Yaskawa INFORM job: aprem2TRJ2.JBI

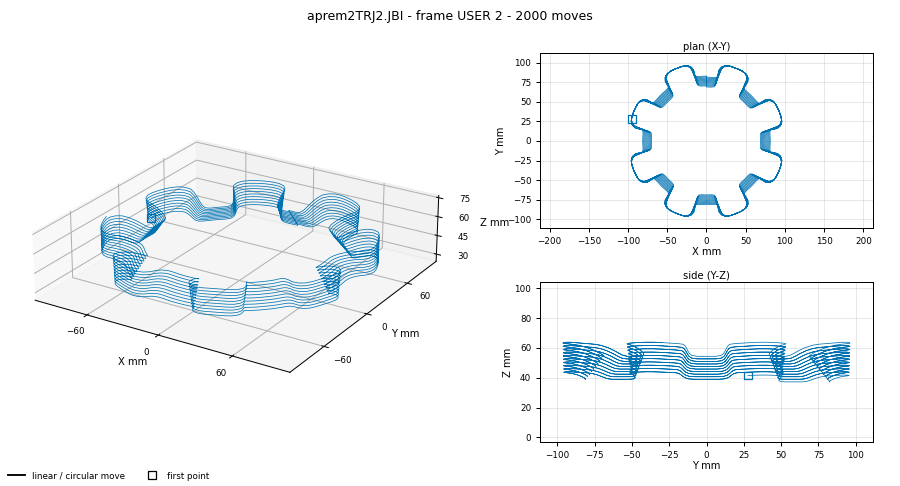
[picture p0: tool path of aprem2TRJ2.JBI in frame USER 2, 2000 of 2000 moves have a stored position in this frame; points joined in program order, loops and branches not executed]
/JOB
//NAME aprem2TRJ2
//POS
///NPOS 2000,0,2000,0,0,0
///USER 2
///TOOL 1
///POSTYPE USER
///RECTAN
///RCONF 1,0,0,0,0,0,0,0,0,0,0,0,0,0,0,0,0,0,0,0,0,0,0,0
C00000=-95.500,27.752,41.515,179.9573,-1.4576,0.0000
C00001=-94.679,31.992,41.678,179.9802,-0.0621,0.0000
C00002=-93.214,36.189,41.785,179.9968,-0.0083,0.0000
C00003=-91.502,40.323,41.785,179.9964,-0.0081,0.0000
C00004=-89.570,44.326,41.678,179.9701,-0.0579,0.0000
C00005=-87.153,47.905,41.515,178.9994,-1.0610,0.0000
C00006=-83.964,50.341,41.355,177.9940,-1.0426,0.0000
C00007=-80.606,51.270,41.159,176.0647,-0.0633,0.0000
C00008=-77.545,50.645,40.789,176.2827,1.1365,0.0000
C00009=-74.511,49.565,40.048,179.1830,0.2954,0.0000
C00010=-71.724,48.673,39.090,-174.7304,-1.4587,0.0000
C00011=-69.261,48.447,38.165,-161.9042,-0.3246,0.0000
C00012=-66.868,49.465,37.495,-150.0988,20.4873,0.0000
C00013=-64.059,52.288,37.229,-152.5931,29.6910,0.0000
C00014=-61.349,55.398,37.217,-152.6199,30.0136,0.0000
C00015=-58.451,58.451,37.225,-151.2604,28.7392,0.0000
C00016=-55.398,61.349,37.217,-149.9866,27.3805,0.0000
C00017=-52.288,64.059,37.229,-150.3100,27.4077,0.0000
C00018=-49.465,66.868,37.495,-159.5118,29.9009,0.0000
C00019=-48.447,69.261,38.165,179.6754,18.0958,0.0000
C00020=-48.673,71.724,39.090,178.5413,5.2696,0.0000
C00021=-49.565,74.511,40.048,-179.7046,-0.8170,0.0000
C00022=-50.645,77.545,40.789,-178.8635,-3.7173,0.0000
C00023=-51.270,80.606,41.159,179.9367,-3.9353,0.0000
C00024=-50.341,83.964,41.355,178.9574,-2.0060,0.0000
C00025=-47.905,87.153,41.515,178.9390,-1.0006,0.0000
C00026=-44.326,89.570,41.678,179.9421,-0.0299,0.0000
C00027=-40.323,91.502,41.785,179.9919,-0.0036,0.0000
C00028=-36.189,93.214,41.785,179.9917,-0.0032,0.0000
C00029=-31.992,94.679,41.678,179.9379,-0.0198,0.0000
C00030=-27.752,95.500,41.515,178.5424,-0.0427,0.0000
C00031=-23.775,94.968,41.355,177.8447,0.6817,0.0000
C00032=-20.743,93.250,41.159,177.1705,2.7402,0.0000
C00033=-19.021,90.644,40.789,178.1721,3.4318,0.0000
C00034=-17.640,87.735,40.048,179.6311,0.7865,0.0000
C00035=-16.299,85.134,39.090,-177.2970,-4.7574,0.0000
C00036=-14.718,83.232,38.165,-167.2077,-13.2282,0.0000
C00037=-12.305,82.260,37.495,-146.1451,-8.1050,0.0000
C00038=-8.324,82.270,37.229,-142.4105,2.0911,0.0000
C00039=-4.208,82.553,37.217,-142.2353,2.4190,0.0000
C00040=0.000,82.662,37.225,-142.2055,0.0004,0.0000
C00041=0.000,81.307,38.958,-141.7581,0.0003,0.0000
C00042=4.084,81.202,38.949,-141.7876,-2.4412,0.0000
C00043=8.115,80.931,38.962,-141.9747,-1.8578,0.0000
C00044=12.050,80.963,39.253,-146.2950,9.3084,0.0000
C00045=14.402,82.041,39.987,-169.0753,12.6711,0.0000
C00046=15.932,84.113,41.004,-178.0957,3.7141,0.0000
C00047=17.234,86.943,42.060,179.2930,-1.6621,0.0000
C00048=18.580,90.119,42.880,177.9599,-4.2630,0.0000
C00049=20.259,92.987,43.289,176.7690,-3.4884,0.0000
C00050=23.317,94.913,43.506,177.4450,-0.9091,0.0000
C00051=27.389,95.566,43.684,178.3657,0.0207,0.0000
C00052=31.762,94.755,43.864,179.9236,0.0242,0.0000
C00053=36.110,93.244,43.984,179.9901,0.0038,0.0000
C00054=40.400,91.468,43.984,179.9903,0.0044,0.0000
C00055=44.543,89.461,43.864,179.9289,0.0369,0.0000
C00056=48.209,86.942,43.684,178.8296,1.1411,0.0000
C00057=50.626,83.601,43.506,178.8351,2.4492,0.0000
C00058=51.426,80.077,43.289,-179.8173,4.7459,0.0000
C00059=50.586,76.861,42.880,-178.4237,4.4542,0.0000
C00060=49.291,73.664,42.060,-179.3244,1.6751,0.0000
C00061=48.211,70.742,41.004,178.7173,-3.9706,0.0000
C00062=47.828,68.195,39.987,178.7113,-16.4605,0.0000
C00063=48.729,65.770,39.253,-160.4159,-30.4372,0.0000
C00064=51.488,62.965,38.962,-150.0628,-27.9244,0.0000
C00065=54.531,60.307,38.949,-149.5942,-27.7685,0.0000
C00066=57.493,57.493,38.958,-150.8703,-29.1301,0.0000
C00067=60.306,54.531,38.949,-152.2311,-30.4055,0.0000
C00068=62.965,51.488,38.962,-152.0747,-29.9361,0.0000
C00069=65.770,48.729,39.253,-149.5629,-19.5850,0.0000
C00070=68.195,47.828,39.987,-163.5395,1.2887,0.0000
C00071=70.742,48.211,41.004,-176.0294,1.2827,0.0000
C00072=73.664,49.291,42.060,178.3249,-0.6756,0.0000
C00073=76.861,50.586,42.880,175.5458,-1.5763,0.0000
C00074=80.077,51.426,43.289,175.2541,-0.1827,0.0000
C00075=83.601,50.626,43.506,177.5508,1.1649,0.0000
C00076=86.942,48.209,43.684,178.8589,1.1704,0.0000
C00077=89.461,44.543,43.864,179.9631,0.0711,0.0000
C00078=91.468,40.400,43.984,179.9956,0.0097,0.0000
C00079=93.244,36.110,43.984,179.9962,0.0099,0.0000
C00080=94.755,31.762,43.864,179.9758,0.0764,0.0000
C00081=95.566,27.389,43.684,179.9793,1.6343,0.0000
C00082=94.913,23.317,43.506,-179.0909,2.5550,0.0000
C00083=92.987,20.259,43.289,-176.5116,3.2310,0.0000
C00084=90.119,18.580,42.880,-175.7370,2.0401,0.0000
C00085=86.943,17.234,42.060,-178.3379,0.7070,0.0000
C00086=84.113,15.932,41.004,176.2859,-1.9043,0.0000
C00087=82.041,14.402,39.987,167.3289,-10.9247,0.0000
C00088=80.963,12.050,39.253,170.6916,-33.7050,0.0000
C00089=80.931,8.115,38.962,-178.1422,-38.0253,0.0000
C00090=81.202,4.084,38.949,-177.5588,-38.2124,0.0000
C00091=81.307,0.000,38.958,179.9997,-38.2419,0.0000
C00092=81.202,-4.084,38.949,177.5593,-38.2124,0.0000
C00093=80.931,-8.116,38.962,178.1440,-38.0251,0.0000
C00094=80.963,-12.050,39.253,-170.6925,-33.7054,0.0000
C00095=82.041,-14.402,39.987,-167.3289,-10.9247,0.0000
C00096=84.113,-15.932,41.004,-176.2859,-1.9043,0.0000
C00097=86.943,-17.234,42.060,178.3379,0.7070,0.0000
C00098=90.119,-18.580,42.880,175.7370,2.0401,0.0000
C00099=92.987,-20.259,43.289,176.5116,3.2310,0.0000
C00100=94.913,-23.317,43.506,179.0909,2.5550,0.0000
C00101=95.566,-27.389,43.684,-179.9793,1.6343,0.0000
C00102=94.755,-31.762,43.864,-179.9758,0.0764,0.0000
C00103=93.244,-36.110,43.984,-179.9962,0.0099,0.0000
C00104=91.468,-40.400,43.984,-179.9956,0.0097,0.0000
C00105=89.461,-44.543,43.864,-179.9631,0.0711,0.0000
C00106=86.942,-48.209,43.684,-178.8589,1.1704,0.0000
C00107=83.601,-50.626,43.506,-177.5508,1.1649,0.0000
C00108=80.077,-51.426,43.289,-175.2541,-0.1827,0.0000
C00109=76.861,-50.586,42.880,-175.5458,-1.5763,0.0000
C00110=73.664,-49.291,42.060,-178.3249,-0.6756,0.0000
C00111=70.742,-48.211,41.004,176.0294,1.2827,0.0000
C00112=68.195,-47.828,39.987,163.5395,1.2887,0.0000
C00113=65.770,-48.729,39.253,149.5628,-19.5841,0.0000
C00114=62.965,-51.488,38.962,152.0756,-29.9372,0.0000
C00115=60.307,-54.531,38.949,152.2315,-30.4058,0.0000
C00116=57.493,-57.493,38.958,150.8699,-29.1297,0.0000
C00117=54.531,-60.306,38.949,149.5945,-27.7689,0.0000
C00118=51.488,-62.965,38.962,150.0639,-27.9253,0.0000
C00119=48.729,-65.770,39.253,160.4150,-30.4371,0.0000
C00120=47.828,-68.195,39.987,-178.7113,-16.4605,0.0000
C00121=48.211,-70.742,41.004,-178.7173,-3.9706,0.0000
C00122=49.291,-73.664,42.060,179.3244,1.6751,0.0000
C00123=50.586,-76.861,42.880,178.4237,4.4542,0.0000
C00124=51.426,-80.077,43.289,179.8173,4.7459,0.0000
C00125=50.626,-83.601,43.506,-178.8351,2.4492,0.0000
C00126=48.209,-86.942,43.684,-178.8296,1.1411,0.0000
C00127=44.543,-89.461,43.864,-179.9289,0.0369,0.0000
C00128=40.400,-91.468,43.984,-179.9903,0.0044,0.0000
C00129=36.110,-93.244,43.984,-179.9901,0.0038,0.0000
C00130=31.762,-94.755,43.864,-179.9236,0.0242,0.0000
C00131=27.389,-95.566,43.684,-178.3657,0.0207,0.0000
C00132=23.317,-94.913,43.506,-177.4450,-0.9091,0.0000
C00133=20.259,-92.987,43.289,-176.7690,-3.4884,0.0000
C00134=18.580,-90.119,42.880,-177.9599,-4.2630,0.0000
C00135=17.234,-86.943,42.060,-179.2930,-1.6621,0.0000
C00136=15.932,-84.113,41.004,178.0957,3.7141,0.0000
C00137=14.402,-82.041,39.987,169.0753,12.6711,0.0000
C00138=12.050,-80.963,39.253,146.2950,9.3084,0.0000
C00139=8.115,-80.931,38.962,141.9747,-1.8578,0.0000
C00140=4.084,-81.202,38.949,141.7876,-2.4412,0.0000
C00141=0.000,-81.307,38.958,141.7581,0.0003,0.0000
C00142=0.000,-81.307,38.958,141.7581,0.0003,0.0000
C00143=-4.084,-81.202,38.949,141.7876,2.4407,0.0000
C00144=-8.116,-80.931,38.962,141.9749,1.8560,0.0000
C00145=-12.050,-80.963,39.253,146.2946,-9.3075,0.0000
C00146=-14.402,-82.041,39.987,169.0753,-12.6711,0.0000
C00147=-15.932,-84.113,41.004,178.0957,-3.7141,0.0000
C00148=-17.234,-86.943,42.060,-179.2930,1.6621,0.0000
C00149=-18.580,-90.119,42.880,-177.9599,4.2630,0.0000
C00150=-20.259,-92.987,43.289,-176.7690,3.4884,0.0000
C00151=-23.317,-94.913,43.506,-177.4450,0.9091,0.0000
C00152=-27.389,-95.566,43.684,-178.3657,-0.0207,0.0000
C00153=-31.762,-94.755,43.864,-179.9236,-0.0242,0.0000
C00154=-36.110,-93.244,43.984,-179.9901,-0.0038,0.0000
C00155=-40.400,-91.468,43.984,-179.9903,-0.0044,0.0000
C00156=-44.543,-89.461,43.864,-179.9289,-0.0369,0.0000
C00157=-48.209,-86.942,43.684,-178.8296,-1.1411,0.0000
C00158=-50.626,-83.601,43.506,-178.8351,-2.4492,0.0000
C00159=-51.426,-80.077,43.289,179.8173,-4.7459,0.0000
C00160=-50.586,-76.861,42.880,178.4237,-4.4542,0.0000
C00161=-49.291,-73.664,42.060,179.3244,-1.6751,0.0000
C00162=-48.211,-70.742,41.004,-178.7173,3.9706,0.0000
C00163=-47.828,-68.195,39.987,-178.7113,16.4605,0.0000
C00164=-48.729,-65.770,39.253,160.4159,30.4372,0.0000
C00165=-51.488,-62.965,38.962,150.0628,27.9244,0.0000
C00166=-54.531,-60.307,38.949,149.5942,27.7685,0.0000
C00167=-57.493,-57.493,38.958,150.8703,29.1301,0.0000
C00168=-60.306,-54.531,38.949,152.2311,30.4055,0.0000
C00169=-62.965,-51.488,38.962,152.0747,29.9361,0.0000
C00170=-65.770,-48.729,39.253,149.5629,19.5850,0.0000
C00171=-68.195,-47.828,39.987,163.5395,-1.2887,0.0000
C00172=-70.742,-48.211,41.004,176.0294,-1.2827,0.0000
C00173=-73.664,-49.291,42.060,-178.3249,0.6756,0.0000
C00174=-76.861,-50.586,42.880,-175.5458,1.5763,0.0000
C00175=-80.077,-51.426,43.289,-175.2541,0.1827,0.0000
C00176=-83.601,-50.626,43.506,-177.5508,-1.1649,0.0000
C00177=-86.942,-48.209,43.684,-178.8589,-1.1704,0.0000
C00178=-89.461,-44.543,43.864,-179.9631,-0.0711,0.0000
C00179=-91.468,-40.400,43.984,-179.9956,-0.0097,0.0000
C00180=-93.244,-36.110,43.984,-179.9962,-0.0099,0.0000
C00181=-94.755,-31.762,43.864,-179.9758,-0.0764,0.0000
C00182=-95.566,-27.389,43.684,-179.9793,-1.6343,0.0000
C00183=-94.913,-23.317,43.506,179.0909,-2.5550,0.0000
C00184=-92.987,-20.259,43.289,176.5116,-3.2310,0.0000
C00185=-90.119,-18.580,42.880,175.7370,-2.0401,0.0000
C00186=-86.943,-17.234,42.060,178.3379,-0.7070,0.0000
C00187=-84.113,-15.932,41.004,-176.2859,1.9043,0.0000
C00188=-82.041,-14.402,39.987,-167.3289,10.9247,0.0000
C00189=-80.963,-12.050,39.253,-170.6916,33.7050,0.0000
C00190=-80.931,-8.115,38.962,178.1422,38.0253,0.0000
C00191=-81.202,-4.084,38.949,177.5588,38.2124,0.0000
C00192=-81.307,0.000,38.958,-179.9997,38.2419,0.0000
C00193=-81.202,4.084,38.949,-177.5593,38.2124,0.0000
C00194=-80.931,8.116,38.962,-178.1440,38.0251,0.0000
C00195=-80.963,12.050,39.253,170.6925,33.7054,0.0000
C00196=-82.041,14.402,39.987,167.3289,10.9247,0.0000
C00197=-84.113,15.932,41.004,176.2859,1.9043,0.0000
C00198=-86.943,17.234,42.060,-178.3379,-0.7070,0.0000
C00199=-90.119,18.580,42.880,-175.7370,-2.0401,0.0000
C00200=-92.987,20.259,43.289,-176.5116,-3.2310,0.0000
C00201=-94.913,23.317,43.506,-179.0909,-2.5550,0.0000
C00202=-95.566,27.389,43.684,179.9793,-1.6343,0.0000
C00203=-94.755,31.762,43.864,179.9758,-0.0764,0.0000
C00204=-93.244,36.110,43.984,179.9962,-0.0099,0.0000
C00205=-91.468,40.400,43.984,179.9956,-0.0097,0.0000
C00206=-89.461,44.543,43.864,179.9631,-0.0711,0.0000
C00207=-86.942,48.209,43.684,178.8589,-1.1704,0.0000
C00208=-83.601,50.626,43.506,177.5508,-1.1649,0.0000
C00209=-80.077,51.426,43.289,175.2541,0.1827,0.0000
C00210=-76.861,50.586,42.880,175.5458,1.5763,0.0000
C00211=-73.664,49.291,42.060,178.3249,0.6756,0.0000
C00212=-70.742,48.211,41.004,-176.0294,-1.2827,0.0000
C00213=-68.195,47.828,39.987,-163.5395,-1.2887,0.0000
C00214=-65.770,48.729,39.253,-149.5628,19.5841,0.0000
C00215=-62.965,51.488,38.962,-152.0756,29.9372,0.0000
C00216=-60.307,54.531,38.949,-152.2315,30.4058,0.0000
C00217=-57.493,57.493,38.958,-150.8699,29.1297,0.0000
C00218=-54.531,60.306,38.949,-149.5945,27.7689,0.0000
C00219=-51.488,62.965,38.962,-150.0639,27.9253,0.0000
C00220=-48.729,65.770,39.253,-160.4150,30.4371,0.0000
C00221=-47.828,68.195,39.987,178.7113,16.4605,0.0000
C00222=-48.211,70.742,41.004,178.7173,3.9706,0.0000
C00223=-49.291,73.664,42.060,-179.3244,-1.6751,0.0000
C00224=-50.586,76.861,42.880,-178.4237,-4.4542,0.0000
C00225=-51.426,80.077,43.289,-179.8173,-4.7459,0.0000
C00226=-50.626,83.601,43.506,178.8351,-2.4492,0.0000
C00227=-48.209,86.942,43.684,178.8296,-1.1411,0.0000
C00228=-44.543,89.461,43.864,179.9289,-0.0369,0.0000
C00229=-40.400,91.468,43.984,179.9903,-0.0044,0.0000
C00230=-36.110,93.244,43.984,179.9901,-0.0038,0.0000
C00231=-31.762,94.755,43.864,179.9236,-0.0242,0.0000
C00232=-27.389,95.566,43.684,178.3657,-0.0207,0.0000
C00233=-23.317,94.913,43.506,177.4450,0.9091,0.0000
C00234=-20.259,92.987,43.289,176.7690,3.4884,0.0000
C00235=-18.580,90.119,42.880,177.9599,4.2630,0.0000
C00236=-17.234,86.943,42.060,179.2930,1.6621,0.0000
C00237=-15.932,84.113,41.004,-178.0957,-3.7141,0.0000
C00238=-14.402,82.041,39.987,-169.0753,-12.6711,0.0000
C00239=-12.050,80.963,39.253,-146.2946,-9.3075,0.0000
C00240=-8.116,80.931,38.962,-141.9749,1.8560,0.0000
C00241=-4.084,81.202,38.949,-141.7876,2.4407,0.0000
C00242=0.000,81.307,38.958,-141.7581,0.0003,0.0000
C00243=0.000,79.940,40.681,-141.3945,0.0003,0.0000
C00244=3.959,79.840,40.672,-141.4236,-2.4543,0.0000
C00245=7.905,79.580,40.686,-141.6255,-1.5989,0.0000
C00246=11.791,79.654,41.003,-146.5959,10.4668,0.0000
C00247=14.083,80.839,41.802,-170.8088,11.8957,0.0000
C00248=15.561,83.082,42.912,-178.7432,2.6994,0.0000
C00249=16.825,86.143,44.068,179.0449,-2.4598,0.0000
C00250=18.134,89.588,44.968,177.8329,-5.0059,0.0000
C00251=19.771,92.721,45.418,176.4774,-4.2024,0.0000
C00252=22.856,94.857,45.657,177.0847,-1.1491,0.0000
C00253=27.022,95.633,45.852,178.2015,-0.0057,0.0000
C00254=31.529,94.831,46.051,179.9101,0.0282,0.0000
C00255=36.031,93.275,46.182,179.9885,0.0043,0.0000
C00256=40.478,91.433,46.182,179.9888,0.0050,0.0000
C00257=44.762,89.350,46.051,179.9165,0.0436,0.0000
C00258=48.515,86.730,45.852,178.7321,1.2760,0.0000
C00259=50.913,83.236,45.657,178.7496,2.8735,0.0000
C00260=51.583,79.544,45.418,-179.5172,5.4544,0.0000
C00261=50.526,76.172,44.968,-177.9852,5.0686,0.0000
C00262=49.015,72.810,44.068,-178.9351,2.4144,0.0000
C00263=47.744,69.752,42.912,178.9787,-2.7968,0.0000
C00264=47.203,67.120,41.802,178.0217,-14.7549,0.0000
C00265=47.986,64.662,41.003,-161.4435,-30.8352,0.0000
C00266=50.682,61.862,40.686,-149.9004,-28.3778,0.0000
C00267=53.655,59.255,40.672,-149.2767,-28.0885,0.0000
C00268=56.526,56.526,40.681,-150.5516,-29.4487,0.0000
C00269=59.255,53.656,40.672,-151.9113,-30.7231,0.0000
C00270=61.862,50.682,40.686,-151.6213,-30.0984,0.0000
C00271=64.662,47.986,41.003,-149.1649,-18.5575,0.0000
C00272=67.120,47.203,41.802,-165.2451,1.9783,0.0000
C00273=69.752,47.744,42.912,-177.2032,1.0213,0.0000
C00274=72.810,49.015,44.068,177.5856,-1.0649,0.0000
C00275=76.172,50.526,44.968,174.9314,-2.0148,0.0000
C00276=79.544,51.583,45.418,174.5456,-0.4828,0.0000
C00277=83.236,50.913,45.657,177.1265,1.2504,0.0000
C00278=86.730,48.515,45.852,178.7240,1.2679,0.0000
C00279=89.350,44.762,46.051,179.9564,0.0835,0.0000
C00280=91.433,40.478,46.182,179.9950,0.0112,0.0000
C00281=93.275,36.031,46.182,179.9957,0.0115,0.0000
C00282=94.831,31.529,46.051,179.9718,0.0899,0.0000
C00283=95.633,27.022,45.852,-179.9943,1.7985,0.0000
C00284=94.857,22.856,45.657,-178.8509,2.9153,0.0000
C00285=92.721,19.771,45.418,-175.7976,3.5226,0.0000
C00286=89.588,18.134,44.968,-174.9941,2.1671,0.0000
C00287=86.143,16.825,44.068,-177.5402,0.9551,0.0000
C00288=83.082,15.561,42.912,177.3006,-1.2568,0.0000
C00289=80.839,14.083,41.802,168.1043,-9.1912,0.0000
C00290=79.654,11.791,41.003,169.5332,-33.4041,0.0000
C00291=79.580,7.905,40.686,-178.4011,-38.3745,0.0000
C00292=79.840,3.959,40.672,-177.5457,-38.5764,0.0000
C00293=79.940,0.000,40.681,179.9997,-38.6055,0.0000
C00294=79.840,-3.959,40.672,177.5462,-38.5764,0.0000
C00295=79.580,-7.905,40.686,178.4031,-38.3743,0.0000
C00296=79.654,-11.792,41.003,-169.5340,-33.4045,0.0000
C00297=80.839,-14.083,41.802,-168.1043,-9.1912,0.0000
C00298=83.082,-15.561,42.912,-177.3006,-1.2568,0.0000
C00299=86.143,-16.825,44.068,177.5402,0.9551,0.0000
C00300=89.588,-18.134,44.968,174.9941,2.1671,0.0000
C00301=92.721,-19.771,45.418,175.7976,3.5226,0.0000
C00302=94.857,-22.856,45.657,178.8509,2.9153,0.0000
C00303=95.633,-27.022,45.852,179.9943,1.7985,0.0000
C00304=94.831,-31.529,46.051,-179.9718,0.0899,0.0000
C00305=93.275,-36.031,46.182,-179.9957,0.0115,0.0000
C00306=91.433,-40.478,46.182,-179.9950,0.0112,0.0000
C00307=89.350,-44.762,46.051,-179.9564,0.0835,0.0000
C00308=86.730,-48.515,45.852,-178.7240,1.2679,0.0000
C00309=83.236,-50.913,45.657,-177.1265,1.2504,0.0000
C00310=79.544,-51.583,45.418,-174.5456,-0.4828,0.0000
C00311=76.172,-50.526,44.968,-174.9314,-2.0148,0.0000
C00312=72.810,-49.015,44.068,-177.5856,-1.0649,0.0000
C00313=69.752,-47.744,42.912,177.2032,1.0213,0.0000
C00314=67.120,-47.203,41.802,165.2451,1.9783,0.0000
C00315=64.662,-47.986,41.003,149.1648,-18.5565,0.0000
C00316=61.862,-50.682,40.686,151.6222,-30.0996,0.0000
C00317=59.255,-53.655,40.672,151.9115,-30.7233,0.0000
C00318=56.526,-56.526,40.681,150.5513,-29.4484,0.0000
C00319=53.656,-59.255,40.672,149.2769,-28.0887,0.0000
C00320=50.682,-61.862,40.686,149.9016,-28.3787,0.0000
C00321=47.986,-64.662,41.003,161.4425,-30.8351,0.0000
C00322=47.203,-67.120,41.802,-178.0217,-14.7549,0.0000
C00323=47.744,-69.752,42.912,-178.9787,-2.7968,0.0000
C00324=49.015,-72.810,44.068,178.9351,2.4144,0.0000
C00325=50.526,-76.172,44.968,177.9852,5.0686,0.0000
C00326=51.583,-79.544,45.418,179.5172,5.4544,0.0000
C00327=50.913,-83.236,45.657,-178.7496,2.8735,0.0000
C00328=48.515,-86.730,45.852,-178.7321,1.2760,0.0000
C00329=44.762,-89.350,46.051,-179.9165,0.0436,0.0000
C00330=40.478,-91.433,46.182,-179.9888,0.0050,0.0000
C00331=36.031,-93.275,46.182,-179.9885,0.0043,0.0000
C00332=31.529,-94.831,46.051,-179.9101,0.0282,0.0000
C00333=27.022,-95.633,45.852,-178.2015,-0.0057,0.0000
C00334=22.856,-94.857,45.657,-177.0847,-1.1491,0.0000
C00335=19.771,-92.721,45.418,-176.4774,-4.2024,0.0000
C00336=18.134,-89.588,44.968,-177.8329,-5.0059,0.0000
C00337=16.825,-86.143,44.068,-179.0449,-2.4598,0.0000
C00338=15.561,-83.082,42.912,178.7432,2.6994,0.0000
C00339=14.083,-80.839,41.802,170.8088,11.8957,0.0000
C00340=11.791,-79.654,41.003,146.5959,10.4668,0.0000
C00341=7.905,-79.580,40.686,141.6255,-1.5989,0.0000
C00342=3.959,-79.840,40.672,141.4236,-2.4543,0.0000
C00343=0.000,-79.940,40.681,141.3945,0.0003,0.0000
C00344=0.000,-79.940,40.681,141.3945,0.0003,0.0000
C00345=-3.959,-79.840,40.672,141.4236,2.4538,0.0000
C00346=-7.905,-79.580,40.686,141.6257,1.5969,0.0000
C00347=-11.792,-79.654,41.003,146.5955,-10.4660,0.0000
C00348=-14.083,-80.839,41.802,170.8088,-11.8957,0.0000
C00349=-15.561,-83.082,42.912,178.7432,-2.6994,0.0000
C00350=-16.825,-86.143,44.068,-179.0449,2.4598,0.0000
C00351=-18.134,-89.588,44.968,-177.8329,5.0059,0.0000
C00352=-19.771,-92.721,45.418,-176.4774,4.2024,0.0000
C00353=-22.856,-94.857,45.657,-177.0847,1.1491,0.0000
C00354=-27.022,-95.633,45.852,-178.2015,0.0057,0.0000
C00355=-31.529,-94.831,46.051,-179.9101,-0.0282,0.0000
C00356=-36.031,-93.275,46.182,-179.9885,-0.0043,0.0000
C00357=-40.478,-91.433,46.182,-179.9888,-0.0050,0.0000
C00358=-44.762,-89.350,46.051,-179.9165,-0.0436,0.0000
C00359=-48.515,-86.730,45.852,-178.7321,-1.2760,0.0000
C00360=-50.913,-83.236,45.657,-178.7496,-2.8735,0.0000
C00361=-51.583,-79.544,45.418,179.5172,-5.4544,0.0000
C00362=-50.526,-76.172,44.968,177.9852,-5.0686,0.0000
C00363=-49.015,-72.810,44.068,178.9351,-2.4144,0.0000
C00364=-47.744,-69.752,42.912,-178.9787,2.7968,0.0000
C00365=-47.203,-67.120,41.802,-178.0217,14.7549,0.0000
C00366=-47.986,-64.662,41.003,161.4435,30.8352,0.0000
C00367=-50.682,-61.862,40.686,149.9004,28.3778,0.0000
C00368=-53.655,-59.255,40.672,149.2767,28.0885,0.0000
C00369=-56.526,-56.526,40.681,150.5516,29.4487,0.0000
C00370=-59.255,-53.656,40.672,151.9113,30.7231,0.0000
C00371=-61.862,-50.682,40.686,151.6213,30.0984,0.0000
C00372=-64.662,-47.986,41.003,149.1649,18.5575,0.0000
C00373=-67.120,-47.203,41.802,165.2451,-1.9783,0.0000
C00374=-69.752,-47.744,42.912,177.2032,-1.0213,0.0000
C00375=-72.810,-49.015,44.068,-177.5856,1.0649,0.0000
C00376=-76.172,-50.526,44.968,-174.9314,2.0148,0.0000
C00377=-79.544,-51.583,45.418,-174.5456,0.4828,0.0000
C00378=-83.236,-50.913,45.657,-177.1265,-1.2504,0.0000
C00379=-86.730,-48.515,45.852,-178.7240,-1.2679,0.0000
C00380=-89.350,-44.762,46.051,-179.9564,-0.0835,0.0000
C00381=-91.433,-40.478,46.182,-179.9950,-0.0112,0.0000
C00382=-93.275,-36.031,46.182,-179.9957,-0.0115,0.0000
C00383=-94.831,-31.529,46.051,-179.9718,-0.0899,0.0000
C00384=-95.633,-27.022,45.852,179.9943,-1.7985,0.0000
C00385=-94.857,-22.856,45.657,178.8509,-2.9153,0.0000
C00386=-92.721,-19.771,45.418,175.7976,-3.5226,0.0000
C00387=-89.588,-18.134,44.968,174.9941,-2.1671,0.0000
C00388=-86.143,-16.825,44.068,177.5402,-0.9551,0.0000
C00389=-83.082,-15.561,42.912,-177.3006,1.2568,0.0000
C00390=-80.839,-14.083,41.802,-168.1043,9.1912,0.0000
C00391=-79.654,-11.791,41.003,-169.5332,33.4041,0.0000
C00392=-79.580,-7.905,40.686,178.4011,38.3745,0.0000
C00393=-79.840,-3.959,40.672,177.5457,38.5764,0.0000
C00394=-79.940,0.000,40.681,-179.9997,38.6055,0.0000
C00395=-79.840,3.959,40.672,-177.5462,38.5764,0.0000
C00396=-79.580,7.905,40.686,-178.4031,38.3743,0.0000
C00397=-79.654,11.792,41.003,169.5340,33.4045,0.0000
C00398=-80.839,14.083,41.802,168.1043,9.1912,0.0000
C00399=-83.082,15.561,42.912,177.3006,1.2568,0.0000
C00400=-86.143,16.825,44.068,-177.5402,-0.9551,0.0000
C00401=-89.588,18.134,44.968,-174.9941,-2.1671,0.0000
C00402=-92.721,19.771,45.418,-175.7976,-3.5226,0.0000
C00403=-94.857,22.856,45.657,-178.8509,-2.9153,0.0000
C00404=-95.633,27.022,45.852,-179.9943,-1.7985,0.0000
C00405=-94.831,31.529,46.051,179.9718,-0.0899,0.0000
C00406=-93.275,36.031,46.182,179.9957,-0.0115,0.0000
C00407=-91.433,40.478,46.182,179.9950,-0.0112,0.0000
C00408=-89.350,44.762,46.051,179.9564,-0.0835,0.0000
C00409=-86.730,48.515,45.852,178.7240,-1.2679,0.0000
C00410=-83.236,50.913,45.657,177.1265,-1.2504,0.0000
C00411=-79.544,51.583,45.418,174.5456,0.4828,0.0000
C00412=-76.172,50.526,44.968,174.9314,2.0148,0.0000
C00413=-72.810,49.015,44.068,177.5856,1.0649,0.0000
C00414=-69.752,47.744,42.912,-177.2032,-1.0213,0.0000
C00415=-67.120,47.203,41.802,-165.2451,-1.9783,0.0000
C00416=-64.662,47.986,41.003,-149.1648,18.5565,0.0000
C00417=-61.862,50.682,40.686,-151.6222,30.0996,0.0000
C00418=-59.255,53.655,40.672,-151.9115,30.7233,0.0000
C00419=-56.526,56.526,40.681,-150.5513,29.4484,0.0000
C00420=-53.656,59.255,40.672,-149.2769,28.0887,0.0000
C00421=-50.682,61.862,40.686,-149.9016,28.3787,0.0000
C00422=-47.986,64.662,41.003,-161.4425,30.8351,0.0000
C00423=-47.203,67.120,41.802,178.0217,14.7549,0.0000
C00424=-47.744,69.752,42.912,178.9787,2.7968,0.0000
C00425=-49.015,72.810,44.068,-178.9351,-2.4144,0.0000
C00426=-50.526,76.172,44.968,-177.9852,-5.0686,0.0000
C00427=-51.583,79.544,45.418,-179.5172,-5.4544,0.0000
C00428=-50.913,83.236,45.657,178.7496,-2.8735,0.0000
C00429=-48.515,86.730,45.852,178.7321,-1.2760,0.0000
C00430=-44.762,89.350,46.051,179.9165,-0.0436,0.0000
C00431=-40.478,91.433,46.182,179.9888,-0.0050,0.0000
C00432=-36.031,93.275,46.182,179.9885,-0.0043,0.0000
C00433=-31.529,94.831,46.051,179.9101,-0.0282,0.0000
C00434=-27.022,95.633,45.852,178.2015,0.0057,0.0000
C00435=-22.856,94.857,45.657,177.0847,1.1491,0.0000
C00436=-19.771,92.721,45.418,176.4774,4.2024,0.0000
C00437=-18.134,89.588,44.968,177.8329,5.0059,0.0000
C00438=-16.825,86.143,44.068,179.0449,2.4598,0.0000
C00439=-15.561,83.082,42.912,-178.7432,-2.6994,0.0000
C00440=-14.083,80.839,41.802,-170.8088,-11.8957,0.0000
C00441=-11.792,79.654,41.003,-146.5955,-10.4660,0.0000
C00442=-7.905,79.580,40.686,-141.6257,1.5969,0.0000
C00443=-3.959,79.840,40.672,-141.4236,2.4538,0.0000
C00444=0.000,79.940,40.681,-141.3945,0.0003,0.0000
C00445=0.000,78.562,42.397,-141.1109,0.0002,0.0000
C00446=3.833,78.467,42.387,-141.1396,-2.4588,0.0000
C00447=7.694,78.220,42.402,-141.3590,-1.3181,0.0000
C00448=11.532,78.336,42.745,-147.0431,11.5605,0.0000
C00449=13.762,79.628,43.611,-172.3770,10.9592,0.0000
C00450=15.189,82.045,44.816,-179.2626,1.7346,0.0000
C00451=16.414,85.339,46.074,178.8680,-3.1755,0.0000
C00452=17.687,89.056,47.055,177.7717,-5.6565,0.0000
C00453=19.281,92.454,47.546,176.2826,-4.8619,0.0000
C00454=22.392,94.802,47.807,176.7679,-1.3940,0.0000
C00455=26.654,95.700,48.020,178.0518,-0.0356,0.0000
C00456=31.296,94.909,48.237,179.8977,0.0319,0.0000
C00457=35.952,93.306,48.381,179.9872,0.0049,0.0000
C00458=40.555,91.399,48.381,179.9875,0.0056,0.0000
C00459=44.981,89.240,48.237,179.9051,0.0498,0.0000
C00460=48.823,86.517,48.020,178.6473,1.4030,0.0000
C00461=51.201,82.869,47.807,178.6983,3.2702,0.0000
C00462=51.741,79.009,47.546,-179.1862,6.0558,0.0000
C00463=50.465,75.478,47.055,-177.5651,5.5716,0.0000
C00464=48.737,71.950,46.074,-178.5531,3.0453,0.0000
C00465=47.275,68.755,44.816,179.2946,-1.7479,0.0000
C00466=46.575,66.037,43.611,177.5785,-13.0378,0.0000
C00467=47.238,63.546,42.745,-162.5779,-31.0935,0.0000
C00468=49.870,60.750,42.402,-149.8188,-28.7683,0.0000
C00469=52.774,58.195,42.387,-149.0312,-28.3421,0.0000
C00470=55.552,55.552,42.397,-150.3022,-29.6980,0.0000
C00471=58.195,52.774,42.387,-151.6576,-30.9686,0.0000
C00472=60.750,49.870,42.402,-151.2308,-30.1799,0.0000
C00473=63.546,47.238,42.745,-148.9065,-17.4230,0.0000
C00474=66.037,46.575,43.611,-166.9622,2.4215,0.0000
C00475=68.755,47.275,44.816,-178.2521,0.7054,0.0000
C00476=71.950,48.737,46.074,176.9547,-1.4469,0.0000
C00477=75.478,50.465,47.055,174.4284,-2.4349,0.0000
C00478=79.009,51.741,47.546,173.9442,-0.8138,0.0000
C00479=82.869,51.201,47.807,176.7298,1.3017,0.0000
C00480=86.517,48.823,48.020,178.5970,1.3527,0.0000
C00481=89.240,44.981,48.237,179.9502,0.0949,0.0000
C00482=91.399,40.555,48.381,179.9944,0.0125,0.0000
C00483=93.306,35.952,48.381,179.9951,0.0128,0.0000
C00484=94.909,31.296,48.237,179.9681,0.1023,0.0000
C00485=95.700,26.654,48.020,-179.9644,1.9482,0.0000
C00486=94.802,22.392,47.807,-178.6060,3.2321,0.0000
C00487=92.454,19.281,47.546,-175.1381,3.7174,0.0000
C00488=89.056,17.687,47.055,-174.3435,2.2283,0.0000
C00489=85.339,16.414,46.074,-176.8245,1.1320,0.0000
C00490=82.045,15.189,44.816,178.2654,-0.7374,0.0000
C00491=79.628,13.762,43.611,169.0408,-7.6230,0.0000
C00492=78.336,11.532,42.745,168.4395,-32.9569,0.0000
C00493=78.220,7.694,42.402,-178.6819,-38.6410,0.0000
C00494=78.467,3.833,42.387,-177.5412,-38.8604,0.0000
C00495=78.562,0.000,42.397,179.9998,-38.8891,0.0000
C00496=78.467,-3.833,42.387,177.5416,-38.8604,0.0000
C00497=78.220,-7.694,42.402,178.6839,-38.6407,0.0000
C00498=78.336,-11.532,42.745,-168.4403,-32.9573,0.0000
C00499=79.628,-13.762,43.611,-169.0408,-7.6230,0.0000
C00500=82.045,-15.189,44.816,-178.2654,-0.7374,0.0000
C00501=85.339,-16.414,46.074,176.8245,1.1320,0.0000
C00502=89.056,-17.687,47.055,174.3435,2.2283,0.0000
C00503=92.454,-19.281,47.546,175.1381,3.7174,0.0000
C00504=94.802,-22.392,47.807,178.6060,3.2321,0.0000
C00505=95.700,-26.654,48.020,179.9644,1.9482,0.0000
C00506=94.909,-31.296,48.237,-179.9681,0.1023,0.0000
C00507=93.306,-35.952,48.381,-179.9951,0.0128,0.0000
C00508=91.399,-40.555,48.381,-179.9944,0.0125,0.0000
C00509=89.240,-44.981,48.237,-179.9502,0.0949,0.0000
C00510=86.517,-48.823,48.020,-178.5970,1.3527,0.0000
C00511=82.869,-51.201,47.807,-176.7298,1.3017,0.0000
C00512=79.009,-51.741,47.546,-173.9442,-0.8138,0.0000
C00513=75.478,-50.465,47.055,-174.4284,-2.4349,0.0000
C00514=71.950,-48.737,46.074,-176.9547,-1.4469,0.0000
C00515=68.755,-47.275,44.816,178.2521,0.7054,0.0000
C00516=66.037,-46.575,43.611,166.9622,2.4215,0.0000
C00517=63.546,-47.238,42.745,148.9065,-17.4221,0.0000
C00518=60.750,-49.870,42.402,151.2317,-30.1812,0.0000
C00519=58.195,-52.774,42.387,151.6579,-30.9688,0.0000
C00520=55.552,-55.552,42.397,150.3020,-29.6978,0.0000
C00521=52.774,-58.195,42.387,149.0314,-28.3424,0.0000
C00522=49.870,-60.750,42.402,149.8201,-28.7692,0.0000
C00523=47.238,-63.546,42.745,162.5770,-31.0935,0.0000
C00524=46.575,-66.037,43.611,-177.5785,-13.0378,0.0000
C00525=47.275,-68.755,44.816,-179.2946,-1.7479,0.0000
C00526=48.737,-71.950,46.074,178.5531,3.0453,0.0000
C00527=50.465,-75.478,47.055,177.5651,5.5716,0.0000
C00528=51.741,-79.009,47.546,179.1862,6.0558,0.0000
C00529=51.201,-82.869,47.807,-178.6983,3.2702,0.0000
C00530=48.823,-86.517,48.020,-178.6473,1.4030,0.0000
C00531=44.981,-89.240,48.237,-179.9051,0.0498,0.0000
C00532=40.555,-91.399,48.381,-179.9875,0.0056,0.0000
C00533=35.952,-93.306,48.381,-179.9872,0.0049,0.0000
C00534=31.296,-94.909,48.237,-179.8977,0.0319,0.0000
C00535=26.654,-95.700,48.020,-178.0518,-0.0356,0.0000
C00536=22.392,-94.802,47.807,-176.7679,-1.3940,0.0000
C00537=19.281,-92.454,47.546,-176.2826,-4.8619,0.0000
C00538=17.687,-89.056,47.055,-177.7717,-5.6565,0.0000
C00539=16.414,-85.339,46.074,-178.8680,-3.1755,0.0000
C00540=15.189,-82.045,44.816,179.2626,1.7346,0.0000
C00541=13.762,-79.628,43.611,172.3770,10.9592,0.0000
C00542=11.532,-78.336,42.745,147.0431,11.5605,0.0000
C00543=7.694,-78.220,42.402,141.3590,-1.3181,0.0000
C00544=3.833,-78.467,42.387,141.1396,-2.4588,0.0000
C00545=0.000,-78.562,42.397,141.1109,0.0002,0.0000
C00546=0.000,-78.562,42.397,141.1109,0.0002,0.0000
C00547=-3.833,-78.467,42.387,141.1396,2.4584,0.0000
C00548=-7.694,-78.220,42.402,141.3593,1.3161,0.0000
C00549=-11.532,-78.336,42.745,147.0427,-11.5597,0.0000
C00550=-13.762,-79.628,43.611,172.3770,-10.9592,0.0000
C00551=-15.189,-82.045,44.816,179.2626,-1.7346,0.0000
C00552=-16.414,-85.339,46.074,-178.8680,3.1755,0.0000
C00553=-17.687,-89.056,47.055,-177.7717,5.6565,0.0000
C00554=-19.281,-92.454,47.546,-176.2826,4.8619,0.0000
C00555=-22.392,-94.802,47.807,-176.7679,1.3940,0.0000
C00556=-26.654,-95.700,48.020,-178.0518,0.0356,0.0000
C00557=-31.296,-94.909,48.237,-179.8977,-0.0319,0.0000
C00558=-35.952,-93.306,48.381,-179.9872,-0.0049,0.0000
C00559=-40.555,-91.399,48.381,-179.9875,-0.0056,0.0000
C00560=-44.981,-89.240,48.237,-179.9051,-0.0498,0.0000
C00561=-48.823,-86.517,48.020,-178.6473,-1.4030,0.0000
C00562=-51.201,-82.869,47.807,-178.6983,-3.2702,0.0000
C00563=-51.741,-79.009,47.546,179.1862,-6.0558,0.0000
C00564=-50.465,-75.478,47.055,177.5651,-5.5716,0.0000
C00565=-48.737,-71.950,46.074,178.5531,-3.0453,0.0000
C00566=-47.275,-68.755,44.816,-179.2946,1.7479,0.0000
C00567=-46.575,-66.037,43.611,-177.5785,13.0378,0.0000
C00568=-47.238,-63.546,42.745,162.5779,31.0935,0.0000
C00569=-49.870,-60.750,42.402,149.8188,28.7683,0.0000
C00570=-52.774,-58.195,42.387,149.0312,28.3421,0.0000
C00571=-55.552,-55.552,42.397,150.3022,29.6980,0.0000
C00572=-58.195,-52.774,42.387,151.6576,30.9686,0.0000
C00573=-60.750,-49.870,42.402,151.2308,30.1799,0.0000
C00574=-63.546,-47.238,42.745,148.9065,17.4230,0.0000
C00575=-66.037,-46.575,43.611,166.9622,-2.4215,0.0000
C00576=-68.755,-47.275,44.816,178.2521,-0.7054,0.0000
C00577=-71.950,-48.737,46.074,-176.9547,1.4469,0.0000
C00578=-75.478,-50.465,47.055,-174.4284,2.4349,0.0000
C00579=-79.009,-51.741,47.546,-173.9442,0.8138,0.0000
C00580=-82.869,-51.201,47.807,-176.7298,-1.3017,0.0000
C00581=-86.517,-48.823,48.020,-178.5970,-1.3527,0.0000
C00582=-89.240,-44.981,48.237,-179.9502,-0.0949,0.0000
C00583=-91.399,-40.555,48.381,-179.9944,-0.0125,0.0000
C00584=-93.306,-35.952,48.381,-179.9951,-0.0128,0.0000
C00585=-94.909,-31.296,48.237,-179.9681,-0.1023,0.0000
C00586=-95.700,-26.654,48.020,179.9644,-1.9482,0.0000
C00587=-94.802,-22.392,47.807,178.6060,-3.2321,0.0000
C00588=-92.454,-19.281,47.546,175.1381,-3.7174,0.0000
C00589=-89.056,-17.687,47.055,174.3435,-2.2283,0.0000
C00590=-85.339,-16.414,46.074,176.8245,-1.1320,0.0000
C00591=-82.045,-15.189,44.816,-178.2654,0.7374,0.0000
C00592=-79.628,-13.762,43.611,-169.0408,7.6230,0.0000
C00593=-78.336,-11.532,42.745,-168.4395,32.9569,0.0000
C00594=-78.220,-7.694,42.402,178.6819,38.6410,0.0000
C00595=-78.467,-3.833,42.387,177.5412,38.8604,0.0000
C00596=-78.562,0.000,42.397,-179.9998,38.8891,0.0000
C00597=-78.467,3.833,42.387,-177.5416,38.8604,0.0000
C00598=-78.220,7.694,42.402,-178.6839,38.6407,0.0000
C00599=-78.336,11.532,42.745,168.4403,32.9573,0.0000
C00600=-79.628,13.762,43.611,169.0408,7.6230,0.0000
C00601=-82.045,15.189,44.816,178.2654,0.7374,0.0000
C00602=-85.339,16.414,46.074,-176.8245,-1.1320,0.0000
C00603=-89.056,17.687,47.055,-174.3435,-2.2283,0.0000
C00604=-92.454,19.281,47.546,-175.1381,-3.7174,0.0000
C00605=-94.802,22.392,47.807,-178.6060,-3.2321,0.0000
C00606=-95.700,26.654,48.020,-179.9644,-1.9482,0.0000
C00607=-94.909,31.296,48.237,179.9681,-0.1023,0.0000
C00608=-93.306,35.952,48.381,179.9951,-0.0128,0.0000
C00609=-91.399,40.555,48.381,179.9944,-0.0125,0.0000
C00610=-89.240,44.981,48.237,179.9502,-0.0949,0.0000
C00611=-86.517,48.823,48.020,178.5970,-1.3527,0.0000
C00612=-82.869,51.201,47.807,176.7298,-1.3017,0.0000
C00613=-79.009,51.741,47.546,173.9442,0.8138,0.0000
C00614=-75.478,50.465,47.055,174.4284,2.4349,0.0000
C00615=-71.950,48.737,46.074,176.9547,1.4469,0.0000
C00616=-68.755,47.275,44.816,-178.2521,-0.7054,0.0000
C00617=-66.037,46.575,43.611,-166.9622,-2.4215,0.0000
C00618=-63.546,47.238,42.745,-148.9065,17.4221,0.0000
C00619=-60.750,49.870,42.402,-151.2317,30.1812,0.0000
C00620=-58.195,52.774,42.387,-151.6579,30.9688,0.0000
C00621=-55.552,55.552,42.397,-150.3020,29.6978,0.0000
C00622=-52.774,58.195,42.387,-149.0314,28.3424,0.0000
C00623=-49.870,60.750,42.402,-149.8201,28.7692,0.0000
C00624=-47.238,63.546,42.745,-162.5770,31.0935,0.0000
C00625=-46.575,66.037,43.611,177.5785,13.0378,0.0000
C00626=-47.275,68.755,44.816,179.2946,1.7479,0.0000
C00627=-48.737,71.950,46.074,-178.5531,-3.0453,0.0000
C00628=-50.465,75.478,47.055,-177.5651,-5.5716,0.0000
C00629=-51.741,79.009,47.546,-179.1862,-6.0558,0.0000
C00630=-51.201,82.869,47.807,178.6983,-3.2702,0.0000
C00631=-48.823,86.517,48.020,178.6473,-1.4030,0.0000
C00632=-44.981,89.240,48.237,179.9051,-0.0498,0.0000
C00633=-40.555,91.399,48.381,179.9875,-0.0056,0.0000
C00634=-35.952,93.306,48.381,179.9872,-0.0049,0.0000
C00635=-31.296,94.909,48.237,179.8977,-0.0319,0.0000
C00636=-26.654,95.700,48.020,178.0518,0.0356,0.0000
C00637=-22.392,94.802,47.807,176.7679,1.3940,0.0000
C00638=-19.281,92.454,47.546,176.2826,4.8619,0.0000
C00639=-17.687,89.056,47.055,177.7717,5.6565,0.0000
C00640=-16.414,85.339,46.074,178.8680,3.1755,0.0000
C00641=-15.189,82.045,44.816,-179.2626,-1.7346,0.0000
C00642=-13.762,79.628,43.611,-172.3770,-10.9592,0.0000
C00643=-11.532,78.336,42.745,-147.0427,-11.5597,0.0000
C00644=-7.694,78.220,42.402,-141.3593,1.3161,0.0000
C00645=-3.833,78.467,42.387,-141.1396,2.4584,0.0000
C00646=0.000,78.562,42.397,-141.1109,0.0002,0.0000
C00647=0.000,77.178,44.107,-140.9045,0.0002,0.0000
C00648=3.707,77.088,44.096,-140.9327,-2.4549,0.0000
C00649=7.481,76.852,44.112,-141.1728,-1.0178,0.0000
C00650=11.270,77.011,44.481,-147.6308,12.5713,0.0000
C00651=13.439,78.412,45.416,-173.7657,9.9143,0.0000
C00652=14.814,81.004,46.718,-179.6749,0.8332,0.0000
C00653=16.001,84.532,48.079,178.7474,-3.8082,0.0000
C00654=17.239,88.522,49.141,177.7605,-6.2141,0.0000
C00655=18.791,92.187,49.674,176.1706,-5.4532,0.0000
C00656=21.929,94.746,49.957,176.4973,-1.6362,0.0000
C00657=26.285,95.767,50.188,177.9187,-0.0678,0.0000
C00658=31.062,94.986,50.423,179.8864,0.0352,0.0000
C00659=35.872,93.336,50.579,179.9859,0.0053,0.0000
C00660=40.633,91.364,50.579,179.9863,0.0062,0.0000
C00661=45.201,89.129,50.423,179.8948,0.0555,0.0000
C00662=49.131,86.304,50.188,178.5759,1.5199,0.0000
C00663=51.489,82.502,49.957,178.6776,3.6323,0.0000
C00664=51.899,78.473,49.674,-178.8443,6.5508,0.0000
C00665=50.405,74.784,49.141,-177.1753,5.9740,0.0000
C00666=48.459,71.088,48.079,-178.1897,3.5780,0.0000
C00667=46.803,67.754,46.718,179.6407,-0.8190,0.0000
C00668=45.943,64.949,45.416,177.3464,-11.3560,0.0000
C00669=46.486,62.424,44.481,-163.8001,-31.2115,0.0000
C00670=49.053,59.633,44.112,-149.8158,-29.0968,0.0000
C00671=51.888,57.130,44.096,-148.8556,-28.5314,0.0000
C00672=54.573,54.573,44.107,-150.1203,-29.8799,0.0000
C00673=57.130,51.888,44.096,-151.4684,-31.1443,0.0000
C00674=59.633,49.053,44.112,-150.9023,-30.1828,0.0000
C00675=62.424,46.486,44.482,-148.7885,-16.2008,0.0000
C00676=64.949,45.943,45.416,-168.6440,2.6536,0.0000
C00677=67.754,46.803,46.718,-179.1810,0.3593,0.0000
C00678=71.088,48.459,48.079,176.4220,-1.8103,0.0000
C00679=74.784,50.405,49.141,174.0260,-2.8247,0.0000
C00680=78.473,51.899,49.674,173.4492,-1.1557,0.0000
C00681=82.502,51.489,49.957,176.3677,1.3224,0.0000
C00682=86.304,49.131,50.188,178.4801,1.4241,0.0000
C00683=89.129,45.201,50.423,179.9445,0.1052,0.0000
C00684=91.364,40.633,50.579,179.9938,0.0137,0.0000
C00685=93.336,35.872,50.579,179.9947,0.0141,0.0000
C00686=94.986,31.062,50.423,179.9648,0.1136,0.0000
C00687=95.767,26.285,50.188,-179.9322,2.0813,0.0000
C00688=94.746,21.929,49.957,-178.3638,3.5027,0.0000
C00689=92.187,18.791,49.674,-174.5468,3.8294,0.0000
C00690=88.522,17.239,49.141,-173.7859,2.2395,0.0000
C00691=84.532,16.001,48.079,-176.1918,1.2526,0.0000
C00692=81.004,14.814,46.718,179.1668,-0.3251,0.0000
C00693=78.412,13.439,45.416,170.0857,-6.2343,0.0000
C00694=77.011,11.270,44.481,167.4287,-32.3692,0.0000
C00695=76.852,7.481,44.112,-178.9822,-38.8272,0.0000
C00696=77.088,3.707,44.096,-177.5451,-39.0673,0.0000
C00697=77.178,0.000,44.107,179.9998,-39.0955,0.0000
C00698=77.088,-3.707,44.096,177.5454,-39.0673,0.0000
C00699=76.852,-7.481,44.112,178.9843,-38.8270,0.0000
C00700=77.011,-11.270,44.482,-167.4294,-32.3697,0.0000
C00701=78.412,-13.439,45.416,-170.0857,-6.2343,0.0000
C00702=81.004,-14.814,46.718,-179.1668,-0.3251,0.0000
C00703=84.532,-16.001,48.079,176.1918,1.2526,0.0000
C00704=88.522,-17.239,49.141,173.7859,2.2395,0.0000
C00705=92.187,-18.791,49.674,174.5468,3.8294,0.0000
C00706=94.746,-21.929,49.957,178.3638,3.5027,0.0000
C00707=95.767,-26.285,50.188,179.9322,2.0813,0.0000
C00708=94.986,-31.062,50.423,-179.9648,0.1136,0.0000
C00709=93.336,-35.872,50.579,-179.9947,0.0141,0.0000
C00710=91.364,-40.633,50.579,-179.9938,0.0137,0.0000
C00711=89.129,-45.201,50.423,-179.9445,0.1052,0.0000
C00712=86.304,-49.131,50.188,-178.4801,1.4241,0.0000
C00713=82.502,-51.489,49.957,-176.3677,1.3224,0.0000
C00714=78.473,-51.899,49.674,-173.4492,-1.1557,0.0000
C00715=74.784,-50.405,49.141,-174.0260,-2.8247,0.0000
C00716=71.088,-48.459,48.079,-176.4220,-1.8103,0.0000
C00717=67.754,-46.803,46.718,179.1810,0.3593,0.0000
C00718=64.949,-45.943,45.416,168.6440,2.6536,0.0000
C00719=62.424,-46.486,44.481,148.7885,-16.1999,0.0000
C00720=59.633,-49.053,44.112,150.9032,-30.1842,0.0000
C00721=57.130,-51.888,44.096,151.4686,-31.1444,0.0000
C00722=54.573,-54.573,44.107,150.1201,-29.8797,0.0000
C00723=51.888,-57.130,44.096,148.8557,-28.5316,0.0000
C00724=49.053,-59.633,44.112,149.8172,-29.0977,0.0000
C00725=46.486,-62.424,44.482,163.7992,-31.2115,0.0000
C00726=45.943,-64.949,45.416,-177.3464,-11.3560,0.0000
C00727=46.803,-67.754,46.718,-179.6407,-0.8190,0.0000
C00728=48.459,-71.088,48.079,178.1897,3.5780,0.0000
C00729=50.405,-74.784,49.141,177.1753,5.9740,0.0000
C00730=51.899,-78.473,49.674,178.8443,6.5508,0.0000
C00731=51.489,-82.502,49.957,-178.6776,3.6323,0.0000
C00732=49.131,-86.304,50.188,-178.5759,1.5199,0.0000
C00733=45.201,-89.129,50.423,-179.8948,0.0555,0.0000
C00734=40.633,-91.364,50.579,-179.9863,0.0062,0.0000
C00735=35.872,-93.336,50.579,-179.9859,0.0053,0.0000
C00736=31.062,-94.986,50.423,-179.8864,0.0352,0.0000
C00737=26.285,-95.767,50.188,-177.9187,-0.0678,0.0000
C00738=21.929,-94.746,49.957,-176.4973,-1.6362,0.0000
C00739=18.791,-92.187,49.674,-176.1706,-5.4532,0.0000
C00740=17.239,-88.522,49.141,-177.7605,-6.2141,0.0000
C00741=16.001,-84.532,48.079,-178.7474,-3.8082,0.0000
C00742=14.814,-81.004,46.718,179.6749,0.8332,0.0000
C00743=13.439,-78.412,45.416,173.7657,9.9143,0.0000
C00744=11.270,-77.011,44.481,147.6308,12.5713,0.0000
C00745=7.481,-76.852,44.112,141.1728,-1.0178,0.0000
C00746=3.707,-77.088,44.096,140.9327,-2.4549,0.0000
C00747=0.000,-77.178,44.107,140.9045,0.0002,0.0000
C00748=0.000,-77.178,44.107,140.9045,0.0002,0.0000
C00749=-3.707,-77.088,44.096,140.9327,2.4546,0.0000
C00750=-7.481,-76.852,44.112,141.1730,1.0157,0.0000
C00751=-11.270,-77.011,44.482,147.6303,-12.5706,0.0000
C00752=-13.439,-78.412,45.416,173.7657,-9.9143,0.0000
C00753=-14.814,-81.004,46.718,179.6749,-0.8332,0.0000
C00754=-16.001,-84.532,48.079,-178.7474,3.8082,0.0000
C00755=-17.239,-88.522,49.141,-177.7605,6.2141,0.0000
C00756=-18.791,-92.187,49.674,-176.1706,5.4532,0.0000
C00757=-21.929,-94.746,49.957,-176.4973,1.6362,0.0000
C00758=-26.285,-95.767,50.188,-177.9187,0.0678,0.0000
C00759=-31.062,-94.986,50.423,-179.8864,-0.0352,0.0000
C00760=-35.872,-93.336,50.579,-179.9859,-0.0053,0.0000
C00761=-40.633,-91.364,50.579,-179.9863,-0.0062,0.0000
C00762=-45.201,-89.129,50.423,-179.8948,-0.0555,0.0000
C00763=-49.131,-86.304,50.188,-178.5759,-1.5199,0.0000
C00764=-51.489,-82.502,49.957,-178.6776,-3.6323,0.0000
C00765=-51.899,-78.473,49.674,178.8443,-6.5508,0.0000
C00766=-50.405,-74.784,49.141,177.1753,-5.9740,0.0000
C00767=-48.459,-71.088,48.079,178.1897,-3.5780,0.0000
C00768=-46.803,-67.754,46.718,-179.6407,0.8190,0.0000
C00769=-45.943,-64.949,45.416,-177.3464,11.3560,0.0000
C00770=-46.486,-62.424,44.481,163.8001,31.2115,0.0000
C00771=-49.053,-59.633,44.112,149.8158,29.0968,0.0000
C00772=-51.888,-57.130,44.096,148.8556,28.5314,0.0000
C00773=-54.573,-54.573,44.107,150.1203,29.8799,0.0000
C00774=-57.130,-51.888,44.096,151.4684,31.1443,0.0000
C00775=-59.633,-49.053,44.112,150.9023,30.1828,0.0000
C00776=-62.424,-46.486,44.482,148.7885,16.2008,0.0000
C00777=-64.949,-45.943,45.416,168.6440,-2.6536,0.0000
C00778=-67.754,-46.803,46.718,179.1810,-0.3593,0.0000
C00779=-71.088,-48.459,48.079,-176.4220,1.8103,0.0000
C00780=-74.784,-50.405,49.141,-174.0260,2.8247,0.0000
C00781=-78.473,-51.899,49.674,-173.4492,1.1557,0.0000
C00782=-82.502,-51.489,49.957,-176.3677,-1.3224,0.0000
C00783=-86.304,-49.131,50.188,-178.4801,-1.4241,0.0000
C00784=-89.129,-45.201,50.423,-179.9445,-0.1052,0.0000
C00785=-91.364,-40.633,50.579,-179.9938,-0.0137,0.0000
C00786=-93.336,-35.872,50.579,-179.9947,-0.0141,0.0000
C00787=-94.986,-31.062,50.423,-179.9648,-0.1136,0.0000
C00788=-95.767,-26.285,50.188,179.9322,-2.0813,0.0000
C00789=-94.746,-21.929,49.957,178.3638,-3.5027,0.0000
C00790=-92.187,-18.791,49.674,174.5468,-3.8294,0.0000
C00791=-88.522,-17.239,49.141,173.7859,-2.2395,0.0000
C00792=-84.532,-16.001,48.079,176.1918,-1.2526,0.0000
C00793=-81.004,-14.814,46.718,-179.1668,0.3251,0.0000
C00794=-78.412,-13.439,45.416,-170.0857,6.2343,0.0000
C00795=-77.011,-11.270,44.481,-167.4287,32.3692,0.0000
C00796=-76.852,-7.481,44.112,178.9822,38.8272,0.0000
C00797=-77.088,-3.707,44.096,177.5451,39.0673,0.0000
C00798=-77.178,0.000,44.107,-179.9998,39.0955,0.0000
C00799=-77.088,3.707,44.096,-177.5454,39.0673,0.0000
C00800=-76.852,7.481,44.112,-178.9843,38.8270,0.0000
C00801=-77.011,11.270,44.482,167.4294,32.3697,0.0000
C00802=-78.412,13.439,45.416,170.0857,6.2343,0.0000
C00803=-81.004,14.814,46.718,179.1668,0.3251,0.0000
C00804=-84.532,16.001,48.079,-176.1918,-1.2526,0.0000
C00805=-88.522,17.239,49.141,-173.7859,-2.2395,0.0000
C00806=-92.187,18.791,49.674,-174.5468,-3.8294,0.0000
C00807=-94.746,21.929,49.957,-178.3638,-3.5027,0.0000
C00808=-95.767,26.285,50.188,-179.9322,-2.0813,0.0000
C00809=-94.986,31.062,50.423,179.9648,-0.1136,0.0000
C00810=-93.336,35.872,50.579,179.9947,-0.0141,0.0000
C00811=-91.364,40.633,50.579,179.9938,-0.0137,0.0000
C00812=-89.129,45.201,50.423,179.9445,-0.1052,0.0000
C00813=-86.304,49.131,50.188,178.4801,-1.4241,0.0000
C00814=-82.502,51.489,49.957,176.3677,-1.3224,0.0000
C00815=-78.473,51.899,49.674,173.4492,1.1557,0.0000
C00816=-74.784,50.405,49.141,174.0260,2.8247,0.0000
C00817=-71.088,48.459,48.079,176.4220,1.8103,0.0000
C00818=-67.754,46.803,46.718,-179.1810,-0.3593,0.0000
C00819=-64.949,45.943,45.416,-168.6440,-2.6536,0.0000
C00820=-62.424,46.486,44.481,-148.7885,16.1999,0.0000
C00821=-59.633,49.053,44.112,-150.9032,30.1842,0.0000
C00822=-57.130,51.888,44.096,-151.4686,31.1444,0.0000
C00823=-54.573,54.573,44.107,-150.1201,29.8797,0.0000
C00824=-51.888,57.130,44.096,-148.8557,28.5316,0.0000
C00825=-49.053,59.633,44.112,-149.8172,29.0977,0.0000
C00826=-46.486,62.424,44.482,-163.7992,31.2115,0.0000
C00827=-45.943,64.949,45.416,177.3464,11.3560,0.0000
C00828=-46.803,67.754,46.718,179.6407,0.8190,0.0000
C00829=-48.459,71.088,48.079,-178.1897,-3.5780,0.0000
C00830=-50.405,74.784,49.141,-177.1753,-5.9740,0.0000
C00831=-51.899,78.473,49.674,-178.8443,-6.5508,0.0000
C00832=-51.489,82.502,49.957,178.6776,-3.6323,0.0000
C00833=-49.131,86.304,50.188,178.5759,-1.5199,0.0000
C00834=-45.201,89.129,50.423,179.8948,-0.0555,0.0000
C00835=-40.633,91.364,50.579,179.9863,-0.0062,0.0000
C00836=-35.872,93.336,50.579,179.9859,-0.0053,0.0000
C00837=-31.062,94.986,50.423,179.8864,-0.0352,0.0000
C00838=-26.285,95.767,50.188,177.9187,0.0678,0.0000
C00839=-21.929,94.746,49.957,176.4973,1.6362,0.0000
C00840=-18.791,92.187,49.674,176.1706,5.4532,0.0000
C00841=-17.239,88.522,49.141,177.7605,6.2141,0.0000
C00842=-16.001,84.532,48.079,178.7474,3.8082,0.0000
C00843=-14.814,81.004,46.718,-179.6749,-0.8332,0.0000
C00844=-13.439,78.412,45.416,-173.7657,-9.9143,0.0000
C00845=-11.270,77.011,44.482,-147.6303,-12.5706,0.0000
C00846=-7.481,76.852,44.112,-141.1730,1.0157,0.0000
C00847=-3.707,77.088,44.096,-140.9327,2.4546,0.0000
C00848=0.000,77.178,44.107,-140.9045,0.0002,0.0000
C00849=0.000,75.789,45.812,-140.7733,0.0001,0.0000
C00850=3.580,75.703,45.801,-140.8009,-2.4427,0.0000
C00851=7.267,75.480,45.818,-141.0649,-0.7003,0.0000
C00852=11.008,75.681,46.215,-148.3523,13.4833,0.0000
C00853=13.116,77.193,47.218,-174.9743,8.8067,0.0000
C00854=14.439,79.961,48.618,-179.9989,0.0032,0.0000
C00855=15.588,83.726,50.084,178.6708,-4.3591,0.0000
C00856=16.791,87.989,51.229,177.7869,-6.6807,0.0000
C00857=18.302,91.921,51.802,176.1277,-5.9675,0.0000
C00858=21.467,94.690,52.107,176.2739,-1.8689,0.0000
C00859=25.919,95.834,52.356,177.8036,-0.1013,0.0000
C00860=30.830,95.062,52.610,179.8764,0.0380,0.0000
C00861=35.794,93.367,52.777,179.9849,0.0057,0.0000
C00862=40.710,91.330,52.777,179.9853,0.0067,0.0000
C00863=45.419,89.019,52.610,179.8857,0.0605,0.0000
C00864=49.437,86.092,52.356,178.5181,1.6250,0.0000
C00865=51.776,82.136,52.107,178.6837,3.9541,0.0000
C00866=52.057,77.939,51.802,-178.5076,6.9431,0.0000
C00867=50.345,74.091,51.229,-176.8234,6.2858,0.0000
C00868=48.181,70.226,50.084,-177.8528,4.0217,0.0000
C00869=46.331,66.751,48.618,179.9986,-0.0031,0.0000
C00870=45.309,63.858,47.218,177.2881,-9.7446,0.0000
C00871=45.731,61.299,46.215,-165.0891,-31.1895,0.0000
C00872=48.234,58.511,45.818,-149.8897,-29.3636,0.0000
C00873=50.999,56.061,45.801,-148.7486,-28.6575,0.0000
C00874=53.591,53.591,45.812,-150.0043,-29.9958,0.0000
C00875=56.061,50.999,45.801,-151.3424,-31.2514,0.0000
C00876=58.511,48.233,45.818,-150.6354,-30.1089,0.0000
C00877=61.299,45.731,46.215,-148.8104,-14.9118,0.0000
C00878=63.858,45.309,47.218,-170.2554,2.7119,0.0000
C00879=66.751,46.331,48.618,-179.9969,0.0014,0.0000
C00880=70.226,48.181,50.084,175.9783,-2.1472,0.0000
C00881=74.091,50.345,51.229,173.7142,-3.1766,0.0000
C00882=77.939,52.057,51.802,173.0569,-1.4924,0.0000
C00883=82.136,51.776,52.107,176.0459,1.3163,0.0000
C00884=86.092,49.437,52.356,178.3750,1.4819,0.0000
C00885=89.019,45.419,52.610,179.9395,0.1143,0.0000
C00886=91.330,40.710,52.777,179.9933,0.0147,0.0000
C00887=93.367,35.794,52.777,179.9943,0.0151,0.0000
C00888=95.062,30.830,52.610,179.9620,0.1236,0.0000
C00889=95.834,25.919,52.356,-179.8987,2.1964,0.0000
C00890=94.690,21.467,52.107,-178.1311,3.7261,0.0000
C00891=91.921,18.302,51.802,-174.0325,3.8723,0.0000
C00892=87.989,16.791,51.229,-173.3193,2.2131,0.0000
C00893=83.726,15.588,50.084,-175.6409,1.3292,0.0000
C00894=79.961,14.439,48.618,179.9968,-0.0011,0.0000
C00895=77.193,13.116,47.218,171.1933,-5.0257,0.0000
C00896=75.681,11.008,46.215,166.5167,-31.6477,0.0000
C00897=75.480,7.267,45.818,-179.2997,-38.9351,0.0000
C00898=75.703,3.580,45.801,-177.5573,-39.1991,0.0000
C00899=75.789,0.000,45.812,179.9999,-39.2267,0.0000
C00900=75.703,-3.580,45.801,177.5575,-39.1992,0.0000
C00901=75.480,-7.267,45.818,179.3020,-38.9348,0.0000
C00902=75.681,-11.008,46.215,-166.5172,-31.6482,0.0000
C00903=77.193,-13.116,47.218,-171.1933,-5.0257,0.0000
C00904=79.961,-14.439,48.618,-179.9968,-0.0011,0.0000
C00905=83.726,-15.588,50.084,175.6409,1.3292,0.0000
C00906=87.989,-16.791,51.229,173.3193,2.2131,0.0000
C00907=91.921,-18.302,51.802,174.0325,3.8723,0.0000
C00908=94.690,-21.467,52.107,178.1311,3.7261,0.0000
C00909=95.834,-25.919,52.356,179.8987,2.1964,0.0000
C00910=95.062,-30.830,52.610,-179.9620,0.1236,0.0000
C00911=93.367,-35.794,52.777,-179.9943,0.0151,0.0000
C00912=91.330,-40.710,52.777,-179.9933,0.0147,0.0000
C00913=89.019,-45.419,52.610,-179.9395,0.1143,0.0000
C00914=86.092,-49.437,52.356,-178.3750,1.4819,0.0000
C00915=82.136,-51.776,52.107,-176.0459,1.3163,0.0000
C00916=77.939,-52.057,51.802,-173.0569,-1.4924,0.0000
C00917=74.091,-50.345,51.229,-173.7142,-3.1766,0.0000
C00918=70.226,-48.181,50.084,-175.9783,-2.1472,0.0000
C00919=66.751,-46.331,48.618,179.9969,0.0014,0.0000
C00920=63.858,-45.309,47.218,170.2554,2.7119,0.0000
C00921=61.299,-45.731,46.215,148.8105,-14.9109,0.0000
C00922=58.511,-48.234,45.818,150.6364,-30.1103,0.0000
C00923=56.061,-50.999,45.801,151.3425,-31.2514,0.0000
C00924=53.591,-53.591,45.812,150.0042,-29.9957,0.0000
C00925=50.999,-56.061,45.801,148.7486,-28.6576,0.0000
C00926=48.233,-58.511,45.818,149.8911,-29.3646,0.0000
C00927=45.731,-61.299,46.215,165.0882,-31.1896,0.0000
C00928=45.309,-63.858,47.218,-177.2881,-9.7446,0.0000
C00929=46.331,-66.751,48.618,-179.9986,-0.0031,0.0000
C00930=48.181,-70.226,50.084,177.8528,4.0217,0.0000
C00931=50.345,-74.091,51.229,176.8234,6.2858,0.0000
C00932=52.057,-77.939,51.802,178.5076,6.9431,0.0000
C00933=51.776,-82.136,52.107,-178.6837,3.9541,0.0000
C00934=49.437,-86.092,52.356,-178.5181,1.6250,0.0000
C00935=45.419,-89.019,52.610,-179.8857,0.0605,0.0000
C00936=40.710,-91.330,52.777,-179.9853,0.0067,0.0000
C00937=35.794,-93.367,52.777,-179.9849,0.0057,0.0000
C00938=30.830,-95.062,52.610,-179.8764,0.0380,0.0000
C00939=25.919,-95.834,52.356,-177.8036,-0.1013,0.0000
C00940=21.467,-94.690,52.107,-176.2739,-1.8689,0.0000
C00941=18.302,-91.921,51.802,-176.1277,-5.9675,0.0000
C00942=16.791,-87.989,51.229,-177.7869,-6.6807,0.0000
C00943=15.588,-83.726,50.084,-178.6708,-4.3591,0.0000
C00944=14.439,-79.961,48.618,179.9989,0.0032,0.0000
C00945=13.116,-77.193,47.218,174.9743,8.8067,0.0000
C00946=11.008,-75.681,46.215,148.3523,13.4833,0.0000
C00947=7.267,-75.480,45.818,141.0649,-0.7003,0.0000
C00948=3.580,-75.703,45.801,140.8009,-2.4427,0.0000
C00949=0.000,-75.789,45.812,140.7733,0.0001,0.0000
C00950=0.000,-75.789,45.812,140.7733,0.0001,0.0000
C00951=-3.580,-75.703,45.801,140.8008,2.4425,0.0000
C00952=-7.267,-75.480,45.818,141.0652,0.6980,0.0000
C00953=-11.008,-75.681,46.215,148.3518,-13.4828,0.0000
C00954=-13.116,-77.193,47.218,174.9743,-8.8067,0.0000
C00955=-14.439,-79.961,48.618,179.9989,-0.0032,0.0000
C00956=-15.588,-83.726,50.084,-178.6708,4.3591,0.0000
C00957=-16.791,-87.989,51.229,-177.7869,6.6807,0.0000
C00958=-18.302,-91.921,51.802,-176.1277,5.9675,0.0000
C00959=-21.467,-94.690,52.107,-176.2739,1.8689,0.0000
C00960=-25.919,-95.834,52.356,-177.8036,0.1013,0.0000
C00961=-30.830,-95.062,52.610,-179.8764,-0.0380,0.0000
C00962=-35.794,-93.367,52.777,-179.9849,-0.0057,0.0000
C00963=-40.710,-91.330,52.777,-179.9853,-0.0067,0.0000
C00964=-45.419,-89.019,52.610,-179.8857,-0.0605,0.0000
C00965=-49.437,-86.092,52.356,-178.5181,-1.6250,0.0000
C00966=-51.776,-82.136,52.107,-178.6837,-3.9541,0.0000
C00967=-52.057,-77.939,51.802,178.5076,-6.9431,0.0000
C00968=-50.345,-74.091,51.229,176.8234,-6.2858,0.0000
C00969=-48.181,-70.226,50.084,177.8528,-4.0217,0.0000
C00970=-46.331,-66.751,48.618,-179.9986,0.0031,0.0000
C00971=-45.309,-63.858,47.218,-177.2881,9.7446,0.0000
C00972=-45.731,-61.299,46.215,165.0891,31.1895,0.0000
C00973=-48.234,-58.511,45.818,149.8897,29.3636,0.0000
C00974=-50.999,-56.061,45.801,148.7486,28.6575,0.0000
C00975=-53.591,-53.591,45.812,150.0043,29.9958,0.0000
C00976=-56.061,-50.999,45.801,151.3424,31.2514,0.0000
C00977=-58.511,-48.233,45.818,150.6354,30.1089,0.0000
C00978=-61.299,-45.731,46.215,148.8104,14.9118,0.0000
C00979=-63.858,-45.309,47.218,170.2554,-2.7119,0.0000
C00980=-66.751,-46.331,48.618,179.9969,-0.0014,0.0000
C00981=-70.226,-48.181,50.084,-175.9783,2.1472,0.0000
C00982=-74.091,-50.345,51.229,-173.7142,3.1766,0.0000
C00983=-77.939,-52.057,51.802,-173.0569,1.4924,0.0000
C00984=-82.136,-51.776,52.107,-176.0459,-1.3163,0.0000
C00985=-86.092,-49.437,52.356,-178.3750,-1.4819,0.0000
C00986=-89.019,-45.419,52.610,-179.9395,-0.1143,0.0000
C00987=-91.330,-40.710,52.777,-179.9933,-0.0147,0.0000
C00988=-93.367,-35.794,52.777,-179.9943,-0.0151,0.0000
C00989=-95.062,-30.830,52.610,-179.9620,-0.1236,0.0000
C00990=-95.834,-25.919,52.356,179.8987,-2.1964,0.0000
C00991=-94.690,-21.467,52.107,178.1311,-3.7261,0.0000
C00992=-91.921,-18.302,51.802,174.0325,-3.8723,0.0000
C00993=-87.989,-16.791,51.229,173.3193,-2.2131,0.0000
C00994=-83.726,-15.588,50.084,175.6409,-1.3292,0.0000
C00995=-79.961,-14.439,48.618,-179.9968,0.0011,0.0000
C00996=-77.193,-13.116,47.218,-171.1933,5.0257,0.0000
C00997=-75.681,-11.008,46.215,-166.5167,31.6477,0.0000
C00998=-75.480,-7.267,45.818,179.2997,38.9351,0.0000
C00999=-75.703,-3.580,45.801,177.5573,39.1991,0.0000
C01000=-75.789,0.000,45.812,-179.9999,39.2267,0.0000
C01001=-75.703,3.580,45.801,-177.5575,39.1992,0.0000
C01002=-75.480,7.267,45.818,-179.3020,38.9348,0.0000
C01003=-75.681,11.008,46.215,166.5172,31.6482,0.0000
C01004=-77.193,13.116,47.218,171.1933,5.0257,0.0000
C01005=-79.961,14.439,48.618,179.9968,0.0011,0.0000
C01006=-83.726,15.588,50.084,-175.6409,-1.3292,0.0000
C01007=-87.989,16.791,51.229,-173.3193,-2.2131,0.0000
C01008=-91.921,18.302,51.802,-174.0325,-3.8723,0.0000
C01009=-94.690,21.467,52.107,-178.1311,-3.7261,0.0000
C01010=-95.834,25.919,52.356,-179.8987,-2.1964,0.0000
C01011=-95.062,30.830,52.610,179.9620,-0.1236,0.0000
C01012=-93.367,35.794,52.777,179.9943,-0.0151,0.0000
C01013=-91.330,40.710,52.777,179.9933,-0.0147,0.0000
C01014=-89.019,45.419,52.610,179.9395,-0.1143,0.0000
C01015=-86.092,49.437,52.356,178.3750,-1.4819,0.0000
C01016=-82.136,51.776,52.107,176.0459,-1.3163,0.0000
C01017=-77.939,52.057,51.802,173.0569,1.4924,0.0000
C01018=-74.091,50.345,51.229,173.7142,3.1766,0.0000
C01019=-70.226,48.181,50.084,175.9783,2.1472,0.0000
C01020=-66.751,46.331,48.618,-179.9969,-0.0014,0.0000
C01021=-63.858,45.309,47.218,-170.2554,-2.7119,0.0000
C01022=-61.299,45.731,46.215,-148.8105,14.9109,0.0000
C01023=-58.511,48.234,45.818,-150.6364,30.1103,0.0000
C01024=-56.061,50.999,45.801,-151.3425,31.2514,0.0000
C01025=-53.591,53.591,45.812,-150.0042,29.9957,0.0000
C01026=-50.999,56.061,45.801,-148.7486,28.6576,0.0000
C01027=-48.233,58.511,45.818,-149.8911,29.3646,0.0000
C01028=-45.731,61.299,46.215,-165.0882,31.1896,0.0000
C01029=-45.309,63.858,47.218,177.2881,9.7446,0.0000
C01030=-46.331,66.751,48.618,179.9986,0.0031,0.0000
C01031=-48.181,70.226,50.084,-177.8528,-4.0217,0.0000
C01032=-50.345,74.091,51.229,-176.8234,-6.2858,0.0000
C01033=-52.057,77.939,51.802,-178.5076,-6.9431,0.0000
C01034=-51.776,82.136,52.107,178.6837,-3.9541,0.0000
C01035=-49.437,86.092,52.356,178.5181,-1.6250,0.0000
C01036=-45.419,89.019,52.610,179.8857,-0.0605,0.0000
C01037=-40.710,91.330,52.777,179.9853,-0.0067,0.0000
C01038=-35.794,93.367,52.777,179.9849,-0.0057,0.0000
C01039=-30.830,95.062,52.610,179.8764,-0.0380,0.0000
C01040=-25.919,95.834,52.356,177.8036,0.1013,0.0000
C01041=-21.467,94.690,52.107,176.2739,1.8689,0.0000
C01042=-18.302,91.921,51.802,176.1277,5.9675,0.0000
C01043=-16.791,87.989,51.229,177.7869,6.6807,0.0000
C01044=-15.588,83.726,50.084,178.6708,4.3591,0.0000
C01045=-14.439,79.961,48.618,-179.9989,-0.0032,0.0000
C01046=-13.116,77.193,47.218,-174.9743,-8.8067,0.0000
C01047=-11.008,75.681,46.215,-148.3518,-13.4828,0.0000
C01048=-7.267,75.480,45.818,-141.0652,0.6980,0.0000
C01049=-3.580,75.703,45.801,-140.8008,2.4425,0.0000
C01050=0.000,75.789,45.812,-140.7733,0.0001,0.0000
C01051=0.000,74.396,47.516,-140.7158,0.0000,0.0000
C01052=3.453,74.315,47.503,-140.7427,-2.4223,0.0000
C01053=7.053,74.105,47.522,-141.0345,-0.3681,0.0000
C01054=10.745,74.349,47.946,-149.1996,14.2839,0.0000
C01055=12.792,75.972,49.019,-176.0111,7.6747,0.0000
C01056=14.064,78.919,50.519,179.7498,-0.7514,0.0000
C01057=15.177,82.922,52.090,178.6288,-4.8303,0.0000
C01058=16.346,87.459,53.317,177.8411,-7.0591,0.0000
C01059=17.816,91.657,53.931,176.1414,-6.4001,0.0000
C01060=21.009,94.635,54.258,176.0979,-2.0860,0.0000
C01061=25.555,95.900,54.525,177.7079,-0.1349,0.0000
C01062=30.600,95.138,54.796,179.8678,0.0404,0.0000
C01063=35.715,93.397,54.976,179.9840,0.0060,0.0000
C01064=40.787,91.296,54.976,179.9844,0.0071,0.0000
C01065=45.636,88.910,54.796,179.8779,0.0649,0.0000
C01066=49.741,85.881,54.525,178.4742,1.7165,0.0000
C01067=52.061,81.773,54.258,178.7124,4.2314,0.0000
C01068=52.213,77.409,53.931,-178.1887,7.2383,0.0000
C01069=50.285,73.401,53.317,-176.5147,6.5160,0.0000
C01070=47.903,69.367,52.090,-177.5476,4.3848,0.0000
C01071=45.859,65.749,50.519,-179.6456,0.7082,0.0000
C01072=44.675,62.766,49.019,177.3675,-8.2277,0.0000
C01073=44.975,60.171,47.946,-166.4231,-31.0292,0.0000
C01074=47.412,57.387,47.522,-150.0390,-29.5687,0.0000
C01075=50.108,54.990,47.503,-148.7091,-28.7213,0.0000
C01076=52.606,52.606,47.516,-149.9535,-30.0466,0.0000
C01077=54.990,50.108,47.503,-151.2786,-31.2909,0.0000
C01078=57.387,47.412,47.522,-150.4303,-29.9595,0.0000
C01079=60.171,44.975,47.946,-148.9707,-13.5777,0.0000
C01080=62.766,44.675,49.019,-171.7723,2.6325,0.0000
C01081=65.749,45.859,50.519,179.2918,-0.3544,0.0000
C01082=69.367,47.903,52.090,175.6152,-2.4524,0.0000
C01083=73.401,50.285,53.317,173.4840,-3.4853,0.0000
C01084=77.409,52.213,53.931,172.7617,-1.8113,0.0000
C01085=81.773,52.061,54.258,175.7686,1.2876,0.0000
C01086=85.881,49.741,54.525,178.2835,1.5258,0.0000
C01087=88.910,45.636,54.796,179.9351,0.1221,0.0000
C01088=91.296,40.787,54.976,179.9929,0.0156,0.0000
C01089=93.397,35.715,54.976,179.9940,0.0160,0.0000
C01090=95.138,30.600,54.796,179.9596,0.1322,0.0000
C01091=95.900,25.555,54.525,-179.8651,2.2921,0.0000
C01092=94.635,21.009,54.258,-177.9140,3.9021,0.0000
C01093=91.657,17.816,53.931,-173.5999,3.8586,0.0000
C01094=87.459,16.346,53.317,-172.9409,2.1589,0.0000
C01095=82.922,15.177,52.090,-175.1697,1.3712,0.0000
C01096=78.919,14.064,50.519,-179.2486,0.2502,0.0000
C01097=75.972,12.792,49.019,172.3253,-3.9889,0.0000
C01098=74.349,10.745,47.946,165.7161,-30.8004,0.0000
C01099=74.105,7.053,47.522,-179.6319,-38.9655,0.0000
C01100=74.315,3.453,47.503,-177.5777,-39.2573,0.0000
C01101=74.396,0.000,47.516,180.0000,-39.2842,0.0000
C01102=74.315,-3.453,47.503,177.5778,-39.2573,0.0000
C01103=74.105,-7.053,47.522,179.6343,-38.9652,0.0000
C01104=74.349,-10.745,47.946,-165.7166,-30.8009,0.0000
C01105=75.972,-12.792,49.019,-172.3253,-3.9889,0.0000
C01106=78.919,-14.064,50.519,179.2486,0.2502,0.0000
C01107=82.922,-15.177,52.090,175.1697,1.3712,0.0000
C01108=87.459,-16.346,53.317,172.9409,2.1589,0.0000
C01109=91.657,-17.816,53.931,173.5999,3.8586,0.0000
C01110=94.635,-21.009,54.258,177.9140,3.9021,0.0000
C01111=95.900,-25.555,54.525,179.8651,2.2921,0.0000
C01112=95.138,-30.600,54.796,-179.9596,0.1322,0.0000
C01113=93.397,-35.715,54.976,-179.9940,0.0160,0.0000
C01114=91.296,-40.787,54.976,-179.9929,0.0156,0.0000
C01115=88.910,-45.636,54.796,-179.9351,0.1221,0.0000
C01116=85.881,-49.741,54.525,-178.2835,1.5258,0.0000
C01117=81.773,-52.061,54.258,-175.7686,1.2876,0.0000
C01118=77.409,-52.213,53.931,-172.7617,-1.8113,0.0000
C01119=73.401,-50.285,53.317,-173.4840,-3.4853,0.0000
C01120=69.367,-47.903,52.090,-175.6152,-2.4524,0.0000
C01121=65.749,-45.859,50.519,-179.2918,-0.3544,0.0000
C01122=62.766,-44.675,49.019,171.7723,2.6325,0.0000
C01123=60.171,-44.975,47.946,148.9708,-13.5769,0.0000
C01124=57.387,-47.412,47.522,150.4313,-29.9610,0.0000
C01125=54.990,-50.108,47.503,151.2787,-31.2909,0.0000
C01126=52.606,-52.606,47.516,149.9534,-30.0465,0.0000
C01127=50.108,-54.990,47.503,148.7091,-28.7214,0.0000
C01128=47.412,-57.387,47.522,150.0405,-29.5697,0.0000
C01129=44.975,-60.171,47.946,166.4223,-31.0293,0.0000
C01130=44.675,-62.766,49.019,-177.3675,-8.2277,0.0000
C01131=45.859,-65.749,50.519,179.6456,0.7082,0.0000
C01132=47.903,-69.367,52.090,177.5476,4.3848,0.0000
C01133=50.285,-73.401,53.317,176.5147,6.5160,0.0000
C01134=52.213,-77.409,53.931,178.1887,7.2383,0.0000
C01135=52.061,-81.773,54.258,-178.7124,4.2314,0.0000
C01136=49.741,-85.881,54.525,-178.4742,1.7165,0.0000
C01137=45.636,-88.910,54.796,-179.8779,0.0649,0.0000
C01138=40.787,-91.296,54.976,-179.9844,0.0071,0.0000
C01139=35.715,-93.397,54.976,-179.9840,0.0060,0.0000
C01140=30.600,-95.138,54.796,-179.8678,0.0404,0.0000
C01141=25.555,-95.900,54.525,-177.7079,-0.1349,0.0000
C01142=21.009,-94.635,54.258,-176.0979,-2.0860,0.0000
C01143=17.816,-91.657,53.931,-176.1414,-6.4001,0.0000
C01144=16.346,-87.459,53.317,-177.8411,-7.0591,0.0000
C01145=15.177,-82.922,52.090,-178.6288,-4.8303,0.0000
C01146=14.064,-78.919,50.519,-179.7498,-0.7514,0.0000
C01147=12.792,-75.972,49.019,176.0111,7.6747,0.0000
C01148=10.745,-74.349,47.946,149.1996,14.2839,0.0000
C01149=7.053,-74.105,47.522,141.0345,-0.3681,0.0000
C01150=3.453,-74.315,47.503,140.7427,-2.4223,0.0000
C01151=0.000,-74.396,47.516,140.7158,0.0000,0.0000
C01152=0.000,-74.396,47.516,140.7158,0.0000,0.0000
C01153=-3.453,-74.315,47.503,140.7427,2.4222,0.0000
C01154=-7.053,-74.105,47.522,141.0348,0.3657,0.0000
C01155=-10.745,-74.349,47.946,149.1991,-14.2834,0.0000
C01156=-12.792,-75.972,49.019,176.0111,-7.6747,0.0000
C01157=-14.064,-78.919,50.519,-179.7498,0.7514,0.0000
C01158=-15.177,-82.922,52.090,-178.6288,4.8303,0.0000
C01159=-16.346,-87.459,53.317,-177.8411,7.0591,0.0000
C01160=-17.816,-91.657,53.931,-176.1414,6.4001,0.0000
C01161=-21.009,-94.635,54.258,-176.0979,2.0860,0.0000
C01162=-25.555,-95.900,54.525,-177.7079,0.1349,0.0000
C01163=-30.600,-95.138,54.796,-179.8678,-0.0404,0.0000
C01164=-35.715,-93.397,54.976,-179.9840,-0.0060,0.0000
C01165=-40.787,-91.296,54.976,-179.9844,-0.0071,0.0000
C01166=-45.636,-88.910,54.796,-179.8779,-0.0649,0.0000
C01167=-49.741,-85.881,54.525,-178.4742,-1.7165,0.0000
C01168=-52.061,-81.773,54.258,-178.7124,-4.2314,0.0000
C01169=-52.213,-77.409,53.931,178.1887,-7.2383,0.0000
C01170=-50.285,-73.401,53.317,176.5147,-6.5160,0.0000
C01171=-47.903,-69.367,52.090,177.5476,-4.3848,0.0000
C01172=-45.859,-65.749,50.519,179.6456,-0.7082,0.0000
C01173=-44.675,-62.766,49.019,-177.3675,8.2277,0.0000
C01174=-44.975,-60.171,47.946,166.4231,31.0292,0.0000
C01175=-47.412,-57.387,47.522,150.0390,29.5687,0.0000
C01176=-50.108,-54.990,47.503,148.7091,28.7213,0.0000
C01177=-52.606,-52.606,47.516,149.9535,30.0466,0.0000
C01178=-54.990,-50.108,47.503,151.2786,31.2909,0.0000
C01179=-57.387,-47.412,47.522,150.4303,29.9595,0.0000
C01180=-60.171,-44.975,47.946,148.9707,13.5777,0.0000
C01181=-62.766,-44.675,49.019,171.7723,-2.6325,0.0000
C01182=-65.749,-45.859,50.519,-179.2918,0.3544,0.0000
C01183=-69.367,-47.903,52.090,-175.6152,2.4524,0.0000
C01184=-73.401,-50.285,53.317,-173.4840,3.4853,0.0000
C01185=-77.409,-52.213,53.931,-172.7617,1.8113,0.0000
C01186=-81.773,-52.061,54.258,-175.7686,-1.2876,0.0000
C01187=-85.881,-49.741,54.525,-178.2835,-1.5258,0.0000
C01188=-88.910,-45.636,54.796,-179.9351,-0.1221,0.0000
C01189=-91.296,-40.787,54.976,-179.9929,-0.0156,0.0000
C01190=-93.397,-35.715,54.976,-179.9940,-0.0160,0.0000
C01191=-95.138,-30.600,54.796,-179.9596,-0.1322,0.0000
C01192=-95.900,-25.555,54.525,179.8651,-2.2921,0.0000
C01193=-94.635,-21.009,54.258,177.9140,-3.9021,0.0000
C01194=-91.657,-17.816,53.931,173.5999,-3.8586,0.0000
C01195=-87.459,-16.346,53.317,172.9409,-2.1589,0.0000
C01196=-82.922,-15.177,52.090,175.1697,-1.3712,0.0000
C01197=-78.919,-14.064,50.519,179.2486,-0.2502,0.0000
C01198=-75.972,-12.792,49.019,-172.3253,3.9889,0.0000
C01199=-74.349,-10.745,47.946,-165.7161,30.8004,0.0000
C01200=-74.105,-7.053,47.522,179.6319,38.9655,0.0000
C01201=-74.315,-3.453,47.503,177.5777,39.2573,0.0000
C01202=-74.396,0.000,47.516,-180.0000,39.2842,0.0000
C01203=-74.315,3.453,47.503,-177.5778,39.2573,0.0000
C01204=-74.105,7.053,47.522,-179.6343,38.9652,0.0000
C01205=-74.349,10.745,47.946,165.7166,30.8009,0.0000
C01206=-75.972,12.792,49.019,172.3253,3.9889,0.0000
C01207=-78.919,14.064,50.519,-179.2486,-0.2502,0.0000
C01208=-82.922,15.177,52.090,-175.1697,-1.3712,0.0000
C01209=-87.459,16.346,53.317,-172.9409,-2.1589,0.0000
C01210=-91.657,17.816,53.931,-173.5999,-3.8586,0.0000
C01211=-94.635,21.009,54.258,-177.9140,-3.9021,0.0000
C01212=-95.900,25.555,54.525,-179.8651,-2.2921,0.0000
C01213=-95.138,30.600,54.796,179.9596,-0.1322,0.0000
C01214=-93.397,35.715,54.976,179.9940,-0.0160,0.0000
C01215=-91.296,40.787,54.976,179.9929,-0.0156,0.0000
C01216=-88.910,45.636,54.796,179.9351,-0.1221,0.0000
C01217=-85.881,49.741,54.525,178.2835,-1.5258,0.0000
C01218=-81.773,52.061,54.258,175.7686,-1.2876,0.0000
C01219=-77.409,52.213,53.931,172.7617,1.8113,0.0000
C01220=-73.401,50.285,53.317,173.4840,3.4853,0.0000
C01221=-69.367,47.903,52.090,175.6152,2.4524,0.0000
C01222=-65.749,45.859,50.519,179.2918,0.3544,0.0000
C01223=-62.766,44.675,49.019,-171.7723,-2.6325,0.0000
C01224=-60.171,44.975,47.946,-148.9708,13.5769,0.0000
C01225=-57.387,47.412,47.522,-150.4313,29.9610,0.0000
C01226=-54.990,50.108,47.503,-151.2787,31.2909,0.0000
C01227=-52.606,52.606,47.516,-149.9534,30.0465,0.0000
C01228=-50.108,54.990,47.503,-148.7091,28.7214,0.0000
C01229=-47.412,57.387,47.522,-150.0405,29.5697,0.0000
C01230=-44.975,60.171,47.946,-166.4223,31.0293,0.0000
C01231=-44.675,62.766,49.019,177.3675,8.2277,0.0000
C01232=-45.859,65.749,50.519,-179.6456,-0.7082,0.0000
C01233=-47.903,69.367,52.090,-177.5476,-4.3848,0.0000
C01234=-50.285,73.401,53.317,-176.5147,-6.5160,0.0000
C01235=-52.213,77.409,53.931,-178.1887,-7.2383,0.0000
C01236=-52.061,81.773,54.258,178.7124,-4.2314,0.0000
C01237=-49.741,85.881,54.525,178.4742,-1.7165,0.0000
C01238=-45.636,88.910,54.796,179.8779,-0.0649,0.0000
C01239=-40.787,91.296,54.976,179.9844,-0.0071,0.0000
C01240=-35.715,93.397,54.976,179.9840,-0.0060,0.0000
C01241=-30.600,95.138,54.796,179.8678,-0.0404,0.0000
C01242=-25.555,95.900,54.525,177.7079,0.1349,0.0000
C01243=-21.009,94.635,54.258,176.0979,2.0860,0.0000
C01244=-17.816,91.657,53.931,176.1414,6.4001,0.0000
C01245=-16.346,87.459,53.317,177.8411,7.0591,0.0000
C01246=-15.177,82.922,52.090,178.6288,4.8303,0.0000
C01247=-14.064,78.919,50.519,179.7498,0.7514,0.0000
C01248=-12.792,75.972,49.019,-176.0111,-7.6747,0.0000
C01249=-10.745,74.349,47.946,-149.1991,-14.2834,0.0000
C01250=-7.053,74.105,47.522,-141.0348,0.3657,0.0000
C01251=-3.453,74.315,47.503,-140.7427,2.4222,0.0000
C01252=0.000,74.396,47.516,-140.7158,0.0000,0.0000
C01253=0.000,73.003,49.219,-140.7316,-0.0001,0.0000
C01254=3.325,72.927,49.205,-140.7578,-2.3938,0.0000
C01255=6.839,72.729,49.225,-141.0811,-0.0240,0.0000
C01256=10.483,73.017,49.677,-150.1638,14.9630,0.0000
C01257=12.469,74.753,50.822,-176.8894,6.5490,0.0000
C01258=13.691,77.880,52.422,179.5579,-1.4288,0.0000
C01259=14.768,82.123,54.099,178.6140,-5.2247,0.0000
C01260=15.905,86.934,55.407,177.9156,-7.3526,0.0000
C01261=17.335,91.395,56.062,176.2006,-6.7488,0.0000
C01262=20.556,94.581,56.410,175.9685,-2.2822,0.0000
C01263=25.196,95.965,56.695,177.6326,-0.1678,0.0000
C01264=30.373,95.213,56.983,179.8606,0.0424,0.0000
C01265=35.638,93.426,57.174,179.9832,0.0063,0.0000
C01266=40.862,91.262,57.174,179.9837,0.0074,0.0000
C01267=45.849,88.802,56.983,179.8715,0.0686,0.0000
C01268=50.042,85.674,56.695,178.4441,1.7930,0.0000
C01269=52.343,81.414,56.410,178.7594,4.4610,0.0000
C01270=52.368,76.884,56.062,-177.8971,7.4427,0.0000
C01271=50.225,72.718,55.407,-176.2521,6.6721,0.0000
C01272=47.627,68.512,54.099,-177.2776,4.6745,0.0000
C01273=45.389,64.750,52.422,-179.3021,1.3229,0.0000
C01274=44.041,61.675,50.822,177.5521,-6.8204,0.0000
C01275=44.219,59.044,49.677,-167.7797,-30.7331,0.0000
C01276=46.591,56.263,49.225,-150.2631,-29.7114,0.0000
C01277=49.216,53.919,49.205,-148.7368,-28.7232,0.0000
C01278=51.621,51.621,49.219,-149.9674,-30.0326,0.0000
C01279=53.919,49.216,49.205,-151.2767,-31.2632,0.0000
C01280=56.263,46.591,49.225,-150.2876,-29.7354,0.0000
C01281=59.044,44.219,49.677,-149.2668,-12.2210,0.0000
C01282=61.675,44.041,50.822,-173.1796,2.4479,0.0000
C01283=64.750,45.389,52.422,178.6771,-0.6979,0.0000
C01284=68.512,47.627,54.099,175.3255,-2.7224,0.0000
C01285=72.718,50.225,55.407,173.3279,-3.7479,0.0000
C01286=76.884,52.368,56.062,172.5573,-2.1029,0.0000
C01287=81.414,52.343,56.410,175.5390,1.2406,0.0000
C01288=85.674,50.042,56.695,178.2070,1.5559,0.0000
C01289=88.802,45.849,56.983,179.9314,0.1285,0.0000
C01290=91.262,40.862,57.174,179.9926,0.0163,0.0000
C01291=93.426,35.638,57.174,179.9937,0.0168,0.0000
C01292=95.213,30.373,56.983,179.9576,0.1394,0.0000
C01293=95.965,25.196,56.695,-179.8322,2.3674,0.0000
C01294=94.581,20.556,56.410,-177.7178,4.0315,0.0000
C01295=91.395,17.335,56.062,-173.2512,3.7994,0.0000
C01296=86.934,15.905,55.407,-172.6474,2.0844,0.0000
C01297=82.123,14.768,54.099,-174.7753,1.3860,0.0000
C01298=77.880,13.691,52.422,-178.5712,0.4421,0.0000
C01299=74.753,12.469,50.822,173.4510,-3.1106,0.0000
C01300=73.017,10.483,49.677,165.0370,-29.8362,0.0000
C01301=72.729,6.839,49.225,-179.9760,-38.9189,0.0000
C01302=72.927,3.325,49.205,-177.6062,-39.2422,0.0000
C01303=73.003,0.000,49.219,-179.9999,-39.2684,0.0000
C01304=72.927,-3.325,49.205,177.6063,-39.2423,0.0000
C01305=72.729,-6.839,49.225,179.9785,-38.9186,0.0000
C01306=73.017,-10.483,49.677,-165.0374,-29.8367,0.0000
C01307=74.753,-12.469,50.822,-173.4510,-3.1106,0.0000
C01308=77.880,-13.691,52.422,178.5712,0.4421,0.0000
C01309=82.123,-14.768,54.099,174.7753,1.3860,0.0000
C01310=86.934,-15.905,55.407,172.6474,2.0844,0.0000
C01311=91.395,-17.335,56.062,173.2512,3.7994,0.0000
C01312=94.581,-20.556,56.410,177.7178,4.0315,0.0000
C01313=95.965,-25.196,56.695,179.8322,2.3674,0.0000
C01314=95.213,-30.373,56.983,-179.9576,0.1394,0.0000
C01315=93.426,-35.638,57.174,-179.9937,0.0168,0.0000
C01316=91.262,-40.862,57.174,-179.9926,0.0163,0.0000
C01317=88.802,-45.849,56.983,-179.9314,0.1285,0.0000
C01318=85.674,-50.042,56.695,-178.2070,1.5559,0.0000
C01319=81.414,-52.343,56.410,-175.5390,1.2406,0.0000
C01320=76.884,-52.368,56.062,-172.5573,-2.1029,0.0000
C01321=72.718,-50.225,55.407,-173.3279,-3.7479,0.0000
C01322=68.512,-47.627,54.099,-175.3255,-2.7224,0.0000
C01323=64.750,-45.389,52.422,-178.6771,-0.6979,0.0000
C01324=61.675,-44.041,50.822,173.1796,2.4479,0.0000
C01325=59.044,-44.219,49.677,149.2669,-12.2203,0.0000
C01326=56.263,-46.591,49.225,150.2886,-29.7369,0.0000
C01327=53.919,-49.216,49.205,151.2768,-31.2632,0.0000
C01328=51.621,-51.621,49.219,149.9674,-30.0326,0.0000
C01329=49.216,-53.919,49.205,148.7368,-28.7233,0.0000
C01330=46.591,-56.263,49.225,150.2646,-29.7124,0.0000
C01331=44.219,-59.044,49.677,167.7790,-30.7332,0.0000
C01332=44.041,-61.675,50.822,-177.5521,-6.8204,0.0000
C01333=45.389,-64.750,52.422,179.3021,1.3229,0.0000
C01334=47.627,-68.512,54.099,177.2776,4.6745,0.0000
C01335=50.225,-72.718,55.407,176.2521,6.6721,0.0000
C01336=52.368,-76.884,56.062,177.8971,7.4427,0.0000
C01337=52.343,-81.414,56.410,-178.7594,4.4610,0.0000
C01338=50.042,-85.674,56.695,-178.4441,1.7930,0.0000
C01339=45.849,-88.802,56.983,-179.8715,0.0686,0.0000
C01340=40.862,-91.262,57.174,-179.9837,0.0074,0.0000
C01341=35.638,-93.426,57.174,-179.9832,0.0063,0.0000
C01342=30.373,-95.213,56.983,-179.8606,0.0424,0.0000
C01343=25.196,-95.965,56.695,-177.6326,-0.1678,0.0000
C01344=20.556,-94.581,56.410,-175.9685,-2.2822,0.0000
C01345=17.335,-91.395,56.062,-176.2006,-6.7488,0.0000
C01346=15.905,-86.934,55.407,-177.9156,-7.3526,0.0000
C01347=14.768,-82.123,54.099,-178.6140,-5.2247,0.0000
C01348=13.691,-77.880,52.422,-179.5579,-1.4288,0.0000
C01349=12.469,-74.753,50.822,176.8894,6.5490,0.0000
C01350=10.483,-73.017,49.677,150.1638,14.9630,0.0000
C01351=6.839,-72.729,49.225,141.0811,-0.0240,0.0000
C01352=3.325,-72.927,49.205,140.7578,-2.3938,0.0000
C01353=0.000,-73.003,49.219,140.7316,-0.0001,0.0000
C01354=0.000,-73.003,49.219,140.7316,-0.0001,0.0000
C01355=-3.325,-72.927,49.205,140.7577,2.3937,0.0000
C01356=-6.839,-72.729,49.225,141.0814,0.0215,0.0000
C01357=-10.483,-73.017,49.677,150.1633,-14.9626,0.0000
C01358=-12.469,-74.753,50.822,176.8894,-6.5490,0.0000
C01359=-13.691,-77.880,52.422,-179.5579,1.4288,0.0000
C01360=-14.768,-82.123,54.099,-178.6140,5.2247,0.0000
C01361=-15.905,-86.934,55.407,-177.9156,7.3526,0.0000
C01362=-17.335,-91.395,56.062,-176.2006,6.7488,0.0000
C01363=-20.556,-94.581,56.410,-175.9685,2.2822,0.0000
C01364=-25.196,-95.965,56.695,-177.6326,0.1678,0.0000
C01365=-30.373,-95.213,56.983,-179.8606,-0.0424,0.0000
C01366=-35.638,-93.426,57.174,-179.9832,-0.0063,0.0000
C01367=-40.862,-91.262,57.174,-179.9837,-0.0074,0.0000
C01368=-45.849,-88.802,56.983,-179.8715,-0.0686,0.0000
C01369=-50.042,-85.674,56.695,-178.4441,-1.7930,0.0000
C01370=-52.343,-81.414,56.410,-178.7594,-4.4610,0.0000
C01371=-52.368,-76.884,56.062,177.8971,-7.4427,0.0000
C01372=-50.225,-72.718,55.407,176.2521,-6.6721,0.0000
C01373=-47.627,-68.512,54.099,177.2776,-4.6745,0.0000
C01374=-45.389,-64.750,52.422,179.3021,-1.3229,0.0000
C01375=-44.041,-61.675,50.822,-177.5521,6.8204,0.0000
C01376=-44.219,-59.044,49.677,167.7797,30.7331,0.0000
C01377=-46.591,-56.263,49.225,150.2631,29.7114,0.0000
C01378=-49.216,-53.919,49.205,148.7368,28.7232,0.0000
C01379=-51.621,-51.621,49.219,149.9674,30.0326,0.0000
C01380=-53.919,-49.216,49.205,151.2767,31.2632,0.0000
C01381=-56.263,-46.591,49.225,150.2876,29.7354,0.0000
C01382=-59.044,-44.219,49.677,149.2668,12.2210,0.0000
C01383=-61.675,-44.041,50.822,173.1796,-2.4479,0.0000
C01384=-64.750,-45.389,52.422,-178.6771,0.6979,0.0000
C01385=-68.512,-47.627,54.099,-175.3255,2.7224,0.0000
C01386=-72.718,-50.225,55.407,-173.3279,3.7479,0.0000
C01387=-76.884,-52.368,56.062,-172.5573,2.1029,0.0000
C01388=-81.414,-52.343,56.410,-175.5390,-1.2406,0.0000
C01389=-85.674,-50.042,56.695,-178.2070,-1.5559,0.0000
C01390=-88.802,-45.849,56.983,-179.9314,-0.1285,0.0000
C01391=-91.262,-40.862,57.174,-179.9926,-0.0163,0.0000
C01392=-93.426,-35.638,57.174,-179.9937,-0.0168,0.0000
C01393=-95.213,-30.373,56.983,-179.9576,-0.1394,0.0000
C01394=-95.965,-25.196,56.695,179.8322,-2.3674,0.0000
C01395=-94.581,-20.556,56.410,177.7178,-4.0315,0.0000
C01396=-91.395,-17.335,56.062,173.2512,-3.7994,0.0000
C01397=-86.934,-15.905,55.407,172.6474,-2.0844,0.0000
C01398=-82.123,-14.768,54.099,174.7753,-1.3860,0.0000
C01399=-77.880,-13.691,52.422,178.5712,-0.4421,0.0000
C01400=-74.753,-12.469,50.822,-173.4510,3.1106,0.0000
C01401=-73.017,-10.483,49.677,-165.0370,29.8362,0.0000
C01402=-72.729,-6.839,49.225,179.9760,38.9189,0.0000
C01403=-72.927,-3.325,49.205,177.6062,39.2422,0.0000
C01404=-73.003,0.000,49.219,179.9999,39.2684,0.0000
C01405=-72.927,3.325,49.205,-177.6063,39.2423,0.0000
C01406=-72.729,6.839,49.225,-179.9785,38.9186,0.0000
C01407=-73.017,10.483,49.677,165.0374,29.8367,0.0000
C01408=-74.753,12.469,50.822,173.4510,3.1106,0.0000
C01409=-77.880,13.691,52.422,-178.5712,-0.4421,0.0000
C01410=-82.123,14.768,54.099,-174.7753,-1.3860,0.0000
C01411=-86.934,15.905,55.407,-172.6474,-2.0844,0.0000
C01412=-91.395,17.335,56.062,-173.2512,-3.7994,0.0000
C01413=-94.581,20.556,56.410,-177.7178,-4.0315,0.0000
C01414=-95.965,25.196,56.695,-179.8322,-2.3674,0.0000
C01415=-95.213,30.373,56.983,179.9576,-0.1394,0.0000
C01416=-93.426,35.638,57.174,179.9937,-0.0168,0.0000
C01417=-91.262,40.862,57.174,179.9926,-0.0163,0.0000
C01418=-88.802,45.849,56.983,179.9314,-0.1285,0.0000
C01419=-85.674,50.042,56.695,178.2070,-1.5559,0.0000
C01420=-81.414,52.343,56.410,175.5390,-1.2406,0.0000
C01421=-76.884,52.368,56.062,172.5573,2.1029,0.0000
C01422=-72.718,50.225,55.407,173.3279,3.7479,0.0000
C01423=-68.512,47.627,54.099,175.3255,2.7224,0.0000
C01424=-64.750,45.389,52.422,178.6771,0.6979,0.0000
C01425=-61.675,44.041,50.822,-173.1796,-2.4479,0.0000
C01426=-59.044,44.219,49.677,-149.2669,12.2203,0.0000
C01427=-56.263,46.591,49.225,-150.2886,29.7369,0.0000
C01428=-53.919,49.216,49.205,-151.2768,31.2632,0.0000
C01429=-51.621,51.621,49.219,-149.9674,30.0326,0.0000
C01430=-49.216,53.919,49.205,-148.7368,28.7233,0.0000
C01431=-46.591,56.263,49.225,-150.2646,29.7124,0.0000
C01432=-44.219,59.044,49.677,-167.7790,30.7332,0.0000
C01433=-44.041,61.675,50.822,177.5521,6.8204,0.0000
C01434=-45.389,64.750,52.422,-179.3021,-1.3229,0.0000
C01435=-47.627,68.512,54.099,-177.2776,-4.6745,0.0000
C01436=-50.225,72.718,55.407,-176.2521,-6.6721,0.0000
C01437=-52.368,76.884,56.062,-177.8971,-7.4427,0.0000
C01438=-52.343,81.414,56.410,178.7594,-4.4610,0.0000
C01439=-50.042,85.674,56.695,178.4441,-1.7930,0.0000
C01440=-45.849,88.802,56.983,179.8715,-0.0686,0.0000
C01441=-40.862,91.262,57.174,179.9837,-0.0074,0.0000
C01442=-35.638,93.426,57.174,179.9832,-0.0063,0.0000
C01443=-30.373,95.213,56.983,179.8606,-0.0424,0.0000
C01444=-25.196,95.965,56.695,177.6326,0.1678,0.0000
C01445=-20.556,94.581,56.410,175.9685,2.2822,0.0000
C01446=-17.335,91.395,56.062,176.2006,6.7488,0.0000
C01447=-15.905,86.934,55.407,177.9156,7.3526,0.0000
C01448=-14.768,82.123,54.099,178.6140,5.2247,0.0000
C01449=-13.691,77.880,52.422,179.5579,1.4288,0.0000
C01450=-12.469,74.753,50.822,-176.8894,-6.5490,0.0000
C01451=-10.483,73.017,49.677,-150.1633,-14.9626,0.0000
C01452=-6.839,72.729,49.225,-141.0814,0.0215,0.0000
C01453=-3.325,72.927,49.205,-140.7577,2.3937,0.0000
C01454=0.000,73.003,49.219,-140.7316,-0.0001,0.0000
C01455=0.000,71.612,50.923,-140.8208,-0.0002,0.0000
C01456=3.198,71.541,50.909,-140.8461,-2.3571,0.0000
C01457=6.625,71.354,50.929,-141.2051,0.3291,0.0000
C01458=10.220,71.688,51.410,-151.2344,15.5138,0.0000
C01459=12.146,73.537,52.627,-177.6255,5.4535,0.0000
C01460=13.319,76.847,54.328,179.4145,-2.0293,0.0000
C01461=14.363,81.331,56.111,178.6204,-5.5448,0.0000
C01462=15.469,86.415,57.500,178.0046,-7.5648,0.0000
C01463=16.861,91.137,58.195,176.2963,-7.0136,0.0000
C01464=20.110,94.527,58.564,175.8846,-2.4532,0.0000
C01465=24.842,96.029,58.865,177.5784,-0.1990,0.0000
C01466=30.149,95.287,59.171,179.8550,0.0439,0.0000
C01467=35.562,93.456,59.373,179.9827,0.0065,0.0000
C01468=40.937,91.230,59.373,179.9831,0.0077,0.0000
C01469=46.059,88.697,59.171,179.8665,0.0715,0.0000
C01470=50.337,85.469,58.865,178.4278,1.8534,0.0000
C01471=52.621,81.060,58.564,178.8209,4.6406,0.0000
C01472=52.521,76.366,58.195,-177.6396,7.5626,0.0000
C01473=50.167,72.043,57.500,-176.0374,6.7604,0.0000
C01474=47.354,67.666,56.111,-177.0453,4.8968,0.0000
C01475=44.921,63.757,54.328,-178.9786,1.8489,0.0000
C01476=43.410,60.587,52.627,177.8131,-5.5306,0.0000
C01477=43.464,57.918,51.410,-169.1369,-30.3048,0.0000
C01478=45.770,55.140,50.929,-150.5612,-29.7906,0.0000
C01479=48.325,52.849,50.909,-148.8319,-28.6632,0.0000
C01480=50.637,50.637,50.923,-150.0461,-29.9537,0.0000
C01481=52.848,48.326,50.909,-151.3368,-31.1682,0.0000
C01482=55.140,45.770,50.930,-150.2084,-29.4371,0.0000
C01483=57.918,43.464,51.410,-149.6951,-10.8637,0.0000
C01484=60.587,43.410,52.627,-174.4694,2.1869,0.0000
C01485=63.757,44.921,54.328,178.1511,-1.0214,0.0000
C01486=67.666,47.354,56.111,175.1032,-2.9547,0.0000
C01487=72.043,50.167,57.500,173.2396,-3.9626,0.0000
C01488=76.366,52.521,58.195,172.4374,-2.3604,0.0000
C01489=81.060,52.621,58.564,175.3594,1.1791,0.0000
C01490=85.469,50.337,58.865,178.1466,1.5722,0.0000
C01491=88.697,46.059,59.171,179.9285,0.1335,0.0000
C01492=91.230,40.937,59.373,179.9923,0.0169,0.0000
C01493=93.456,35.562,59.373,179.9935,0.0173,0.0000
C01494=95.287,30.149,59.171,179.9561,0.1450,0.0000
C01495=96.029,24.842,58.865,-179.8010,2.4216,0.0000
C01496=94.527,20.110,58.564,-177.5468,4.1154,0.0000
C01497=91.137,16.861,58.195,-172.9864,3.7037,0.0000
C01498=86.415,15.469,57.500,-172.4352,1.9954,0.0000
C01499=81.331,14.363,56.111,-174.4552,1.3796,0.0000
C01500=76.847,13.319,54.328,-177.9707,0.5855,0.0000
C01501=73.537,12.146,52.627,174.5465,-2.3745,0.0000
C01502=71.688,10.220,51.410,164.4862,-28.7656,0.0000
C01503=71.354,6.625,50.929,179.6709,-38.7949,0.0000
C01504=71.541,3.198,50.909,-177.6429,-39.1539,0.0000
C01505=71.612,0.000,50.923,-179.9998,-39.1792,0.0000
C01506=71.541,-3.198,50.909,177.6428,-39.1539,0.0000
C01507=71.354,-6.626,50.930,-179.6684,-38.7945,0.0000
C01508=71.688,-10.221,51.410,-164.4865,-28.7660,0.0000
C01509=73.537,-12.146,52.627,-174.5465,-2.3745,0.0000
C01510=76.847,-13.319,54.328,177.9707,0.5855,0.0000
C01511=81.331,-14.363,56.111,174.4552,1.3796,0.0000
C01512=86.415,-15.469,57.500,172.4352,1.9954,0.0000
C01513=91.137,-16.861,58.195,172.9864,3.7037,0.0000
C01514=94.527,-20.110,58.564,177.5468,4.1154,0.0000
C01515=96.029,-24.842,58.865,179.8010,2.4216,0.0000
C01516=95.287,-30.149,59.171,-179.9561,0.1450,0.0000
C01517=93.456,-35.562,59.373,-179.9935,0.0173,0.0000
C01518=91.230,-40.937,59.373,-179.9923,0.0169,0.0000
C01519=88.697,-46.059,59.171,-179.9285,0.1335,0.0000
C01520=85.469,-50.337,58.865,-178.1466,1.5722,0.0000
C01521=81.060,-52.621,58.564,-175.3594,1.1791,0.0000
C01522=76.366,-52.521,58.195,-172.4374,-2.3604,0.0000
C01523=72.043,-50.167,57.500,-173.2396,-3.9626,0.0000
C01524=67.666,-47.354,56.111,-175.1032,-2.9547,0.0000
C01525=63.757,-44.921,54.328,-178.1511,-1.0214,0.0000
C01526=60.587,-43.410,52.627,174.4694,2.1869,0.0000
C01527=57.918,-43.464,51.410,149.6952,-10.8631,0.0000
C01528=55.140,-45.770,50.929,150.2094,-29.4388,0.0000
C01529=52.849,-48.325,50.909,151.3368,-31.1681,0.0000
C01530=50.637,-50.637,50.923,150.0463,-29.9539,0.0000
C01531=48.326,-52.848,50.909,148.8318,-28.6632,0.0000
C01532=45.770,-55.140,50.930,150.5629,-29.7916,0.0000
C01533=43.464,-57.918,51.410,169.1363,-30.3049,0.0000
C01534=43.410,-60.587,52.627,-177.8131,-5.5306,0.0000
C01535=44.921,-63.757,54.328,178.9786,1.8489,0.0000
C01536=47.354,-67.666,56.111,177.0453,4.8968,0.0000
C01537=50.167,-72.043,57.500,176.0374,6.7604,0.0000
C01538=52.521,-76.366,58.195,177.6396,7.5626,0.0000
C01539=52.621,-81.060,58.564,-178.8209,4.6406,0.0000
C01540=50.337,-85.469,58.865,-178.4278,1.8534,0.0000
C01541=46.059,-88.697,59.171,-179.8665,0.0715,0.0000
C01542=40.937,-91.230,59.373,-179.9831,0.0077,0.0000
C01543=35.562,-93.456,59.373,-179.9827,0.0065,0.0000
C01544=30.149,-95.287,59.171,-179.8550,0.0439,0.0000
C01545=24.842,-96.029,58.865,-177.5784,-0.1990,0.0000
C01546=20.110,-94.527,58.564,-175.8846,-2.4532,0.0000
C01547=16.861,-91.137,58.195,-176.2963,-7.0136,0.0000
C01548=15.469,-86.415,57.500,-178.0046,-7.5648,0.0000
C01549=14.363,-81.331,56.111,-178.6204,-5.5448,0.0000
C01550=13.319,-76.847,54.328,-179.4145,-2.0293,0.0000
C01551=12.146,-73.537,52.627,177.6255,5.4535,0.0000
C01552=10.220,-71.688,51.410,151.2344,15.5138,0.0000
C01553=6.625,-71.354,50.929,141.2051,0.3291,0.0000
C01554=3.198,-71.541,50.909,140.8461,-2.3571,0.0000
C01555=0.000,-71.612,50.923,140.8208,-0.0002,0.0000
C01556=0.000,-71.612,50.923,140.8208,-0.0002,0.0000
C01557=-3.198,-71.541,50.909,140.8461,2.3572,0.0000
C01558=-6.626,-71.354,50.930,141.2055,-0.3316,0.0000
C01559=-10.221,-71.688,51.410,151.2340,-15.5135,0.0000
C01560=-12.146,-73.537,52.627,177.6255,-5.4535,0.0000
C01561=-13.319,-76.847,54.328,-179.4145,2.0293,0.0000
C01562=-14.363,-81.331,56.111,-178.6204,5.5448,0.0000
C01563=-15.469,-86.415,57.500,-178.0046,7.5648,0.0000
C01564=-16.861,-91.137,58.195,-176.2963,7.0136,0.0000
C01565=-20.110,-94.527,58.564,-175.8846,2.4532,0.0000
C01566=-24.842,-96.029,58.865,-177.5784,0.1990,0.0000
C01567=-30.149,-95.287,59.171,-179.8550,-0.0439,0.0000
C01568=-35.562,-93.456,59.373,-179.9827,-0.0065,0.0000
C01569=-40.937,-91.230,59.373,-179.9831,-0.0077,0.0000
C01570=-46.059,-88.697,59.171,-179.8665,-0.0715,0.0000
C01571=-50.337,-85.469,58.865,-178.4278,-1.8534,0.0000
C01572=-52.621,-81.060,58.564,-178.8209,-4.6406,0.0000
C01573=-52.521,-76.366,58.195,177.6396,-7.5626,0.0000
C01574=-50.167,-72.043,57.500,176.0374,-6.7604,0.0000
C01575=-47.354,-67.666,56.111,177.0453,-4.8968,0.0000
C01576=-44.921,-63.757,54.328,178.9786,-1.8489,0.0000
C01577=-43.410,-60.587,52.627,-177.8131,5.5306,0.0000
C01578=-43.464,-57.918,51.410,169.1369,30.3048,0.0000
C01579=-45.770,-55.140,50.929,150.5612,29.7906,0.0000
C01580=-48.325,-52.849,50.909,148.8319,28.6632,0.0000
C01581=-50.637,-50.637,50.923,150.0461,29.9537,0.0000
C01582=-52.848,-48.326,50.909,151.3368,31.1682,0.0000
C01583=-55.140,-45.770,50.930,150.2084,29.4371,0.0000
C01584=-57.918,-43.464,51.410,149.6951,10.8637,0.0000
C01585=-60.587,-43.410,52.627,174.4694,-2.1869,0.0000
C01586=-63.757,-44.921,54.328,-178.1511,1.0214,0.0000
C01587=-67.666,-47.354,56.111,-175.1032,2.9547,0.0000
C01588=-72.043,-50.167,57.500,-173.2396,3.9626,0.0000
C01589=-76.366,-52.521,58.195,-172.4374,2.3604,0.0000
C01590=-81.060,-52.621,58.564,-175.3594,-1.1791,0.0000
C01591=-85.469,-50.337,58.865,-178.1466,-1.5722,0.0000
C01592=-88.697,-46.059,59.171,-179.9285,-0.1335,0.0000
C01593=-91.230,-40.937,59.373,-179.9923,-0.0169,0.0000
C01594=-93.456,-35.562,59.373,-179.9935,-0.0173,0.0000
C01595=-95.287,-30.149,59.171,-179.9561,-0.1450,0.0000
C01596=-96.029,-24.842,58.865,179.8010,-2.4216,0.0000
C01597=-94.527,-20.110,58.564,177.5468,-4.1154,0.0000
C01598=-91.137,-16.861,58.195,172.9864,-3.7037,0.0000
C01599=-86.415,-15.469,57.500,172.4352,-1.9954,0.0000
C01600=-81.331,-14.363,56.111,174.4552,-1.3796,0.0000
C01601=-76.847,-13.319,54.328,177.9707,-0.5855,0.0000
C01602=-73.537,-12.146,52.627,-174.5465,2.3745,0.0000
C01603=-71.688,-10.220,51.410,-164.4862,28.7656,0.0000
C01604=-71.354,-6.625,50.929,-179.6709,38.7949,0.0000
C01605=-71.541,-3.198,50.909,177.6429,39.1539,0.0000
C01606=-71.612,0.000,50.923,179.9998,39.1792,0.0000
C01607=-71.541,3.198,50.909,-177.6428,39.1539,0.0000
C01608=-71.354,6.626,50.930,179.6684,38.7945,0.0000
C01609=-71.688,10.221,51.410,164.4865,28.7660,0.0000
C01610=-73.537,12.146,52.627,174.5465,2.3745,0.0000
C01611=-76.847,13.319,54.328,-177.9707,-0.5855,0.0000
C01612=-81.331,14.363,56.111,-174.4552,-1.3796,0.0000
C01613=-86.415,15.469,57.500,-172.4352,-1.9954,0.0000
C01614=-91.137,16.861,58.195,-172.9864,-3.7037,0.0000
C01615=-94.527,20.110,58.564,-177.5468,-4.1154,0.0000
C01616=-96.029,24.842,58.865,-179.8010,-2.4216,0.0000
C01617=-95.287,30.149,59.171,179.9561,-0.1450,0.0000
C01618=-93.456,35.562,59.373,179.9935,-0.0173,0.0000
C01619=-91.230,40.937,59.373,179.9923,-0.0169,0.0000
C01620=-88.697,46.059,59.171,179.9285,-0.1335,0.0000
C01621=-85.469,50.337,58.865,178.1466,-1.5722,0.0000
C01622=-81.060,52.621,58.564,175.3594,-1.1791,0.0000
C01623=-76.366,52.521,58.195,172.4374,2.3604,0.0000
C01624=-72.043,50.167,57.500,173.2396,3.9626,0.0000
C01625=-67.666,47.354,56.111,175.1032,2.9547,0.0000
C01626=-63.757,44.921,54.328,178.1511,1.0214,0.0000
C01627=-60.587,43.410,52.627,-174.4694,-2.1869,0.0000
C01628=-57.918,43.464,51.410,-149.6952,10.8631,0.0000
C01629=-55.140,45.770,50.929,-150.2094,29.4388,0.0000
C01630=-52.849,48.325,50.909,-151.3368,31.1681,0.0000
C01631=-50.637,50.637,50.923,-150.0463,29.9539,0.0000
C01632=-48.326,52.848,50.909,-148.8318,28.6632,0.0000
C01633=-45.770,55.140,50.930,-150.5629,29.7916,0.0000
C01634=-43.464,57.918,51.410,-169.1363,30.3049,0.0000
C01635=-43.410,60.587,52.627,177.8131,5.5306,0.0000
C01636=-44.921,63.757,54.328,-178.9786,-1.8489,0.0000
C01637=-47.354,67.666,56.111,-177.0453,-4.8968,0.0000
C01638=-50.167,72.043,57.500,-176.0374,-6.7604,0.0000
C01639=-52.521,76.366,58.195,-177.6396,-7.5626,0.0000
C01640=-52.621,81.060,58.564,178.8209,-4.6406,0.0000
C01641=-50.337,85.469,58.865,178.4278,-1.8534,0.0000
C01642=-46.059,88.697,59.171,179.8665,-0.0715,0.0000
C01643=-40.937,91.230,59.373,179.9831,-0.0077,0.0000
C01644=-35.562,93.456,59.373,179.9827,-0.0065,0.0000
C01645=-30.149,95.287,59.171,179.8550,-0.0439,0.0000
C01646=-24.842,96.029,58.865,177.5784,0.1990,0.0000
C01647=-20.110,94.527,58.564,175.8846,2.4532,0.0000
C01648=-16.861,91.137,58.195,176.2963,7.0136,0.0000
C01649=-15.469,86.415,57.500,178.0046,7.5648,0.0000
C01650=-14.363,81.331,56.111,178.6204,5.5448,0.0000
C01651=-13.319,76.847,54.328,179.4145,2.0293,0.0000
C01652=-12.146,73.537,52.627,-177.6255,-5.4535,0.0000
C01653=-10.221,71.688,51.410,-151.2340,-15.5135,0.0000
C01654=-6.626,71.354,50.930,-141.2055,-0.3316,0.0000
C01655=-3.198,71.541,50.909,-140.8461,2.3572,0.0000
C01656=0.000,71.612,50.923,-140.8208,-0.0002,0.0000
C01657=0.000,70.224,52.630,-140.9842,-0.0003,0.0000
C01658=3.072,70.158,52.615,-141.0087,-2.3123,0.0000
C01659=6.412,69.984,52.637,-141.4077,0.6880,0.0000
C01660=9.959,70.362,53.146,-152.3999,15.9321,0.0000
C01661=11.825,72.328,54.436,-178.2362,4.4065,0.0000
C01662=12.951,75.822,56.240,179.3107,-2.5537,0.0000
C01663=13.963,80.549,58.128,178.6435,-5.7936,0.0000
C01664=15.041,85.905,59.597,178.1039,-7.6987,0.0000
C01665=16.396,90.884,60.330,176.4208,-7.1953,0.0000
C01666=19.672,94.474,60.719,175.8447,-2.5954,0.0000
C01667=24.496,96.092,61.037,177.5461,-0.2275,0.0000
C01668=29.931,95.359,61.359,179.8510,0.0449,0.0000
C01669=35.488,93.484,61.571,179.9823,0.0066,0.0000
C01670=41.009,91.197,61.571,179.9828,0.0078,0.0000
C01671=46.265,88.593,61.359,179.8629,0.0736,0.0000
C01672=50.626,85.269,61.037,178.4250,1.8965,0.0000
C01673=52.893,80.714,60.719,178.8932,4.7688,0.0000
C01674=52.671,75.858,60.330,-177.4212,7.6040,0.0000
C01675=50.109,71.379,59.597,-175.8716,6.7862,0.0000
C01676=47.084,66.830,58.128,-176.8518,5.0569,0.0000
C01677=44.457,62.772,56.240,-178.6807,2.2931,0.0000
C01678=42.782,59.505,54.436,178.1262,-4.3612,0.0000
C01679=42.712,56.796,53.146,-170.4736,-29.7489,0.0000
C01680=44.952,54.020,52.637,-150.9334,-29.8046,0.0000
C01681=47.437,51.781,52.615,-148.9950,-28.5406,0.0000
C01682=49.656,49.656,52.630,-150.1903,-29.8094,0.0000
C01683=51.781,47.437,52.615,-151.4594,-31.0052,0.0000
C01684=54.020,44.952,52.637,-150.1944,-29.0648,0.0000
C01685=56.796,42.711,53.146,-150.2510,-9.5269,0.0000
C01686=59.505,42.782,54.436,-175.6388,1.8738,0.0000
C01687=62.772,44.457,56.240,177.7069,-1.3193,0.0000
C01688=66.830,47.084,58.128,174.9431,-3.1482,0.0000
C01689=71.379,50.109,59.597,173.2138,-4.1284,0.0000
C01690=75.858,52.671,60.330,172.3960,-2.5788,0.0000
C01691=80.714,52.893,60.719,175.2312,1.1068,0.0000
C01692=85.269,50.626,61.037,178.1035,1.5750,0.0000
C01693=88.593,46.265,61.359,179.9264,0.1371,0.0000
C01694=91.197,41.009,61.571,179.9922,0.0172,0.0000
C01695=93.484,35.488,61.571,179.9934,0.0177,0.0000
C01696=95.359,29.931,61.359,179.9551,0.1490,0.0000
C01697=96.092,24.496,61.037,-179.7725,2.4539,0.0000
C01698=94.474,19.672,60.719,-177.4046,4.1553,0.0000
C01699=90.884,16.396,60.330,-172.8047,3.5792,0.0000
C01700=85.905,15.041,59.597,-172.3013,1.8961,0.0000
C01701=80.549,13.963,58.128,-174.2064,1.3565,0.0000
C01702=75.822,12.951,56.240,-177.4463,0.6893,0.0000
C01703=72.328,11.825,54.436,175.5935,-1.7638,0.0000
C01704=70.362,9.959,53.146,164.0679,-27.6001,0.0000
C01705=69.984,6.412,52.637,179.3120,-38.5923,0.0000
C01706=70.158,3.072,52.615,-177.6877,-38.9913,0.0000
C01707=70.224,0.000,52.630,-179.9997,-39.0158,0.0000
C01708=70.158,-3.071,52.615,177.6875,-38.9914,0.0000
C01709=69.984,-6.412,52.637,-179.3094,-38.5919,0.0000
C01710=70.362,-9.959,53.146,-164.0682,-27.6005,0.0000
C01711=72.328,-11.825,54.436,-175.5935,-1.7638,0.0000
C01712=75.822,-12.951,56.240,177.4463,0.6893,0.0000
C01713=80.549,-13.963,58.128,174.2064,1.3565,0.0000
C01714=85.905,-15.041,59.597,172.3013,1.8961,0.0000
C01715=90.884,-16.396,60.330,172.8047,3.5792,0.0000
C01716=94.474,-19.672,60.719,177.4046,4.1553,0.0000
C01717=96.092,-24.496,61.037,179.7725,2.4539,0.0000
C01718=95.359,-29.931,61.359,-179.9551,0.1490,0.0000
C01719=93.484,-35.488,61.571,-179.9934,0.0177,0.0000
C01720=91.197,-41.009,61.571,-179.9922,0.0172,0.0000
C01721=88.593,-46.265,61.359,-179.9264,0.1371,0.0000
C01722=85.269,-50.626,61.037,-178.1035,1.5750,0.0000
C01723=80.714,-52.893,60.719,-175.2312,1.1068,0.0000
C01724=75.858,-52.671,60.330,-172.3960,-2.5788,0.0000
C01725=71.379,-50.109,59.597,-173.2138,-4.1284,0.0000
C01726=66.830,-47.084,58.128,-174.9431,-3.1482,0.0000
C01727=62.772,-44.457,56.240,-177.7069,-1.3193,0.0000
C01728=59.505,-42.782,54.436,175.6388,1.8738,0.0000
C01729=56.796,-42.712,53.146,150.2511,-9.5264,0.0000
C01730=54.020,-44.952,52.637,150.1954,-29.0666,0.0000
C01731=51.781,-47.437,52.615,151.4594,-31.0050,0.0000
C01732=49.656,-49.656,52.630,150.1906,-29.8097,0.0000
C01733=47.437,-51.781,52.615,148.9948,-28.5406,0.0000
C01734=44.952,-54.020,52.637,150.9352,-29.8056,0.0000
C01735=42.711,-56.796,53.146,170.4731,-29.7490,0.0000
C01736=42.782,-59.505,54.436,-178.1262,-4.3612,0.0000
C01737=44.457,-62.772,56.240,178.6807,2.2931,0.0000
C01738=47.084,-66.830,58.128,176.8518,5.0569,0.0000
C01739=50.109,-71.379,59.597,175.8716,6.7862,0.0000
C01740=52.671,-75.858,60.330,177.4212,7.6040,0.0000
C01741=52.893,-80.714,60.719,-178.8932,4.7688,0.0000
C01742=50.626,-85.269,61.037,-178.4250,1.8965,0.0000
C01743=46.265,-88.593,61.359,-179.8629,0.0736,0.0000
C01744=41.009,-91.197,61.571,-179.9828,0.0078,0.0000
C01745=35.488,-93.484,61.571,-179.9823,0.0066,0.0000
C01746=29.931,-95.359,61.359,-179.8510,0.0449,0.0000
C01747=24.496,-96.092,61.037,-177.5461,-0.2275,0.0000
C01748=19.672,-94.474,60.719,-175.8447,-2.5954,0.0000
C01749=16.396,-90.884,60.330,-176.4208,-7.1953,0.0000
C01750=15.041,-85.905,59.597,-178.1039,-7.6987,0.0000
C01751=13.963,-80.549,58.128,-178.6435,-5.7936,0.0000
C01752=12.951,-75.822,56.240,-179.3107,-2.5537,0.0000
C01753=11.825,-72.328,54.436,178.2362,4.4065,0.0000
C01754=9.959,-70.362,53.146,152.3999,15.9321,0.0000
C01755=6.412,-69.984,52.637,141.4077,0.6880,0.0000
C01756=3.072,-70.158,52.615,141.0087,-2.3123,0.0000
C01757=0.000,-70.224,52.630,140.9842,-0.0003,0.0000
C01758=0.000,-70.224,52.630,140.9842,-0.0003,0.0000
C01759=-3.071,-70.158,52.615,141.0086,2.3125,0.0000
C01760=-6.412,-69.984,52.637,141.4081,-0.6906,0.0000
C01761=-9.959,-70.362,53.146,152.3995,-15.9318,0.0000
C01762=-11.825,-72.328,54.436,178.2362,-4.4065,0.0000
C01763=-12.951,-75.822,56.240,-179.3107,2.5537,0.0000
C01764=-13.963,-80.549,58.128,-178.6435,5.7936,0.0000
C01765=-15.041,-85.905,59.597,-178.1039,7.6987,0.0000
C01766=-16.396,-90.884,60.330,-176.4208,7.1953,0.0000
C01767=-19.672,-94.474,60.719,-175.8447,2.5954,0.0000
C01768=-24.496,-96.092,61.037,-177.5461,0.2275,0.0000
C01769=-29.931,-95.359,61.359,-179.8510,-0.0449,0.0000
C01770=-35.488,-93.484,61.571,-179.9823,-0.0066,0.0000
C01771=-41.009,-91.197,61.571,-179.9828,-0.0078,0.0000
C01772=-46.265,-88.593,61.359,-179.8629,-0.0736,0.0000
C01773=-50.626,-85.269,61.037,-178.4250,-1.8965,0.0000
C01774=-52.893,-80.714,60.719,-178.8932,-4.7688,0.0000
C01775=-52.671,-75.858,60.330,177.4212,-7.6040,0.0000
C01776=-50.109,-71.379,59.597,175.8716,-6.7862,0.0000
C01777=-47.084,-66.830,58.128,176.8518,-5.0569,0.0000
C01778=-44.457,-62.772,56.240,178.6807,-2.2931,0.0000
C01779=-42.782,-59.505,54.436,-178.1262,4.3612,0.0000
C01780=-42.712,-56.796,53.146,170.4736,29.7489,0.0000
C01781=-44.952,-54.020,52.637,150.9334,29.8046,0.0000
C01782=-47.437,-51.781,52.615,148.9950,28.5406,0.0000
C01783=-49.656,-49.656,52.630,150.1903,29.8094,0.0000
C01784=-51.781,-47.437,52.615,151.4594,31.0052,0.0000
C01785=-54.020,-44.952,52.637,150.1944,29.0648,0.0000
C01786=-56.796,-42.711,53.146,150.2510,9.5269,0.0000
C01787=-59.505,-42.782,54.436,175.6388,-1.8738,0.0000
C01788=-62.772,-44.457,56.240,-177.7069,1.3193,0.0000
C01789=-66.830,-47.084,58.128,-174.9431,3.1482,0.0000
C01790=-71.379,-50.109,59.597,-173.2138,4.1284,0.0000
C01791=-75.858,-52.671,60.330,-172.3960,2.5788,0.0000
C01792=-80.714,-52.893,60.719,-175.2312,-1.1068,0.0000
C01793=-85.269,-50.626,61.037,-178.1035,-1.5750,0.0000
C01794=-88.593,-46.265,61.359,-179.9264,-0.1371,0.0000
C01795=-91.197,-41.009,61.571,-179.9922,-0.0172,0.0000
C01796=-93.484,-35.488,61.571,-179.9934,-0.0177,0.0000
C01797=-95.359,-29.931,61.359,-179.9551,-0.1490,0.0000
C01798=-96.092,-24.496,61.037,179.7725,-2.4539,0.0000
C01799=-94.474,-19.672,60.719,177.4046,-4.1553,0.0000
C01800=-90.884,-16.396,60.330,172.8047,-3.5792,0.0000
C01801=-85.905,-15.041,59.597,172.3013,-1.8961,0.0000
C01802=-80.549,-13.963,58.128,174.2064,-1.3565,0.0000
C01803=-75.822,-12.951,56.240,177.4463,-0.6893,0.0000
C01804=-72.328,-11.825,54.436,-175.5935,1.7638,0.0000
C01805=-70.362,-9.959,53.146,-164.0679,27.6001,0.0000
C01806=-69.984,-6.412,52.637,-179.3120,38.5923,0.0000
C01807=-70.158,-3.072,52.615,177.6877,38.9913,0.0000
C01808=-70.224,0.000,52.630,179.9997,39.0158,0.0000
C01809=-70.158,3.071,52.615,-177.6875,38.9914,0.0000
C01810=-69.984,6.412,52.637,179.3094,38.5919,0.0000
C01811=-70.362,9.959,53.146,164.0682,27.6005,0.0000
C01812=-72.328,11.825,54.436,175.5935,1.7638,0.0000
C01813=-75.822,12.951,56.240,-177.4463,-0.6893,0.0000
C01814=-80.549,13.963,58.128,-174.2064,-1.3565,0.0000
C01815=-85.905,15.041,59.597,-172.3013,-1.8961,0.0000
C01816=-90.884,16.396,60.330,-172.8047,-3.5792,0.0000
C01817=-94.474,19.672,60.719,-177.4046,-4.1553,0.0000
C01818=-96.092,24.496,61.037,-179.7725,-2.4539,0.0000
C01819=-95.359,29.931,61.359,179.9551,-0.1490,0.0000
C01820=-93.484,35.488,61.571,179.9934,-0.0177,0.0000
C01821=-91.197,41.009,61.571,179.9922,-0.0172,0.0000
C01822=-88.593,46.265,61.359,179.9264,-0.1371,0.0000
C01823=-85.269,50.626,61.037,178.1035,-1.5750,0.0000
C01824=-80.714,52.893,60.719,175.2312,-1.1068,0.0000
C01825=-75.858,52.671,60.330,172.3960,2.5788,0.0000
C01826=-71.379,50.109,59.597,173.2138,4.1284,0.0000
C01827=-66.830,47.084,58.128,174.9431,3.1482,0.0000
C01828=-62.772,44.457,56.240,177.7069,1.3193,0.0000
C01829=-59.505,42.782,54.436,-175.6388,-1.8738,0.0000
C01830=-56.796,42.712,53.146,-150.2511,9.5264,0.0000
C01831=-54.020,44.952,52.637,-150.1954,29.0666,0.0000
C01832=-51.781,47.437,52.615,-151.4594,31.0050,0.0000
C01833=-49.656,49.656,52.630,-150.1906,29.8097,0.0000
C01834=-47.437,51.781,52.615,-148.9948,28.5406,0.0000
C01835=-44.952,54.020,52.637,-150.9352,29.8056,0.0000
C01836=-42.711,56.796,53.146,-170.4731,29.7490,0.0000
C01837=-42.782,59.505,54.436,178.1262,4.3612,0.0000
C01838=-44.457,62.772,56.240,-178.6807,-2.2931,0.0000
C01839=-47.084,66.830,58.128,-176.8518,-5.0569,0.0000
C01840=-50.109,71.379,59.597,-175.8716,-6.7862,0.0000
C01841=-52.671,75.858,60.330,-177.4212,-7.6040,0.0000
C01842=-52.893,80.714,60.719,178.8932,-4.7688,0.0000
C01843=-50.626,85.269,61.037,178.4250,-1.8965,0.0000
C01844=-46.265,88.593,61.359,179.8629,-0.0736,0.0000
C01845=-41.009,91.197,61.571,179.9828,-0.0078,0.0000
C01846=-35.488,93.484,61.571,179.9823,-0.0066,0.0000
C01847=-29.931,95.359,61.359,179.8510,-0.0449,0.0000
C01848=-24.496,96.092,61.037,177.5461,0.2275,0.0000
C01849=-19.672,94.474,60.719,175.8447,2.5954,0.0000
C01850=-16.396,90.884,60.330,176.4208,7.1953,0.0000
C01851=-15.041,85.905,59.597,178.1039,7.6987,0.0000
C01852=-13.963,80.549,58.128,178.6435,5.7936,0.0000
C01853=-12.951,75.822,56.240,179.3107,2.5537,0.0000
C01854=-11.825,72.328,54.436,-178.2362,-4.4065,0.0000
C01855=-9.959,70.362,53.146,-152.3995,-15.9318,0.0000
C01856=-6.412,69.984,52.637,-141.4081,-0.6906,0.0000
C01857=-3.071,70.158,52.615,-141.0086,2.3125,0.0000
C01858=0.000,70.224,52.630,-140.9842,-0.0003,0.0000
C01859=0.000,68.843,54.342,-141.2235,-0.0004,0.0000
C01860=2.945,68.781,54.326,-141.2470,-2.2595,0.0000
C01861=6.200,68.619,54.350,-141.6907,1.0492,0.0000
C01862=9.699,69.044,54.888,-153.6475,16.2162,0.0000
C01863=11.507,71.127,56.252,-178.7377,3.4210,0.0000
C01864=12.586,74.809,58.158,179.2393,-3.0039,0.0000
C01865=13.569,79.780,60.151,178.6797,-5.9734,0.0000
C01866=14.621,85.405,61.698,178.2099,-7.7575,0.0000
C01867=15.942,90.636,62.469,176.5679,-7.2955,0.0000
C01868=19.246,94.423,62.877,175.8470,-2.7058,0.0000
C01869=24.159,96.154,63.210,177.5359,-0.2528,0.0000
C01870=29.718,95.429,63.547,179.8486,0.0454,0.0000
C01871=35.416,93.512,63.770,179.9821,0.0067,0.0000
C01872=41.080,91.166,63.770,179.9826,0.0079,0.0000
C01873=46.465,88.493,63.547,179.8609,0.0749,0.0000
C01874=50.908,85.074,63.210,178.4357,1.9214,0.0000
C01875=53.158,80.376,62.877,178.9730,4.8449,0.0000
